# B&R Automation Studio project NAEUL004C00R13L518F00 (part 3)

### IoMap.iom - X20CP0483/IoMap.iom
```iecst
VAR_CONFIG
	::AWOpen:bModuleOK AT %IX."AutoWidth".ModuleOk;
	::AWOpen:tyParamInDriver.uiErrCode_603F AT %IW."AutoWidth".ErrorCode_603F;
	::AWOpen:tyParamOutDriver.uiCtrlword_6040 AT %QW."AutoWidth".Controlword_6040;
	::AWOpen:tyParamInDriver.uiStatword_6041 AT %IW."AutoWidth".Statusword_6041;
	::AWOpen:tyParamOutDriver.siModOfOpt_6060 AT %QB."AutoWidth".ModesOfOperation_6060;
	::AWOpen:tyParamInDriver.siModOfOptDisp_6061 AT %IB."AutoWidth".ModesOfOperationDisplay_6061;
	::AWOpen:tyParamInDriver.diActualPos_6064 AT %ID."AutoWidth".PositionActualValue_6064;
	::AWOpen:tyParamOutDriver.diTargetPos_607A AT %QD."AutoWidth".TargetPosition_607A;
	::AWOpen:tyParamOutDriver.udiMoveSpd_6081 AT %QD."AutoWidth".ProfileVelocity_6081;
	::AWOpen:tyParamOutDriver.siHmMethod_6098 AT %QB."AutoWidth".HomingMethod_6098;
	::AWOpen:tyParamInDriver.udiDigitalInputs_60FD AT %ID."AutoWidth".DigitalInputs_60FD;
	::AWOpen:tyParamOutDriver.diJogVel_60FF AT %QD."AutoWidth".TargetVelocity_60FF;
	::LifterBtm:bModuleOK AT %IX."Lifter".ModuleOk;
	::LifterBtm:tyParamInDriver.uiErrCode_603F AT %IW."Lifter".ErrorCode_603F;
	::LifterBtm:tyParamOutDriver.uiCtrlword_6040 AT %QW."Lifter".Controlword_6040;
	::LifterBtm:tyParamInDriver.uiStatword_6041 AT %IW."Lifter".Statusword_6041;
	::LifterBtm:tyParamOutDriver.siModOfOpt_6060 AT %QB."Lifter".ModesOfOperation_6060;
	::LifterBtm:tyParamInDriver.siModOfOptDisp_6061 AT %IB."Lifter".ModesOfOperationDisplay_6061;
	::LifterBtm:tyParamInDriver.diActualPos_6064 AT %ID."Lifter".PositionActualValue_6064;
	::LifterBtm:tyParamOutDriver.diTargetPos_607A AT %QD."Lifter".TargetPosition_607A;
	::LifterBtm:tyParamOutDriver.udiMoveSpd_6081 AT %QD."Lifter".ProfileVelocity_6081;
	::LifterBtm:tyParamOutDriver.siHmMethod_6098 AT %QB."Lifter".HomingMethod_6098;
	::LifterBtm:tyParamInDriver.udiDigitalInputs_60FD AT %ID."Lifter".DigitalInputs_60FD;
	::LifterBtm:tyParamOutDriver.diJogVel_60FF AT %QD."Lifter".TargetVelocity_60FF;
	::Trav:bModuleOK AT %IX."Traverser".ModuleOk;
	::Trav:tyParamInDriver.uiErrCode_603F AT %IW."Traverser".ErrorCode_603F;
	::Trav:tyParamOutDriver.uiCtrlword_6040 AT %QW."Traverser".Controlword_6040;
	::Trav:tyParamInDriver.uiStatword_6041 AT %IW."Traverser".Statusword_6041;
	::Trav:tyParamOutDriver.siModOfOpt_6060 AT %QB."Traverser".ModesOfOperation_6060;
	::Trav:tyParamInDriver.siModOfOptDisp_6061 AT %IB."Traverser".ModesOfOperationDisplay_6061;
	::Trav:tyParamInDriver.diActualPos_6064 AT %ID."Traverser".PositionActualValue_6064;
	::Trav:tyParamOutDriver.diTargetPos_607A AT %QD."Traverser".TargetPosition_607A;
	::Trav:tyParamOutDriver.udiMoveSpd_6081 AT %QD."Traverser".ProfileVelocity_6081;
	::Trav:tyParamOutDriver.siHmMethod_6098 AT %QB."Traverser".HomingMethod_6098;
	::Trav:tyParamInDriver.udiDigitalInputs_60FD AT %ID."Traverser".DigitalInputs_60FD;
	::Trav:tyParamOutDriver.diJogVel_60FF AT %QD."Traverser".TargetVelocity_60FF;
	::DInput:a_bPhysicalDI[1] AT %IX."X20DI9372".DigitalInput01;
	::DInput:a_bPhysicalDI[2] AT %IX."X20DI9372".DigitalInput02;
	::DInput:a_bPhysicalDI[3] AT %IX."X20DI9372".DigitalInput03;
	::DInput:a_bPhysicalDI[4] AT %IX."X20DI9372".DigitalInput04;
	::DInput:a_bPhysicalDI[5] AT %IX."X20DI9372".DigitalInput05;
	::DInput:a_bPhysicalDI[6] AT %IX."X20DI9372".DigitalInput06;
	::DInput:a_bPhysicalDI[7] AT %IX."X20DI9372".DigitalInput07;
	::DInput:a_bPhysicalDI[8] AT %IX."X20DI9372".DigitalInput08;
	::DInput:a_bPhysicalDI[9] AT %IX."X20DI9372".DigitalInput09;
	::DInput:a_bPhysicalDI[10] AT %IX."X20DI9372".DigitalInput10;
	::DInput:a_bPhysicalDI[11] AT %IX."X20DI9372".DigitalInput11;
	::DInput:a_bPhysicalDI[12] AT %IX."X20DI9372".DigitalInput12;
	::DInput:a_bPhysicalDI[13] AT %IX."X20DI9372a".DigitalInput01;
	::DInput:a_bPhysicalDI[14] AT %IX."X20DI9372a".DigitalInput02;
	::DInput:a_bPhysicalDI[15] AT %IX."X20DI9372a".DigitalInput03;
	::DInput:a_bPhysicalDI[16] AT %IX."X20DI9372a".DigitalInput04;
	::DInput:a_bPhysicalDI[17] AT %IX."X20DI9372a".DigitalInput05;
	::DInput:a_bPhysicalDI[18] AT %IX."X20DI9372a".DigitalInput06;
	::DInput:a_bPhysicalDI[19] AT %IX."X20DI9372a".DigitalInput07;
	::DInput:a_bPhysicalDI[20] AT %IX."X20DI9372a".DigitalInput08;
	::DInput:a_bPhysicalDI[21] AT %IX."X20DI9372a".DigitalInput09;
	::DInput:a_bPhysicalDI[22] AT %IX."X20DI9372a".DigitalInput10;
	::DInput:a_bPhysicalDI[23] AT %IX."X20DI9372a".DigitalInput11;
	::DInput:a_bPhysicalDI[24] AT %IX."X20DI9372a".DigitalInput12;
	::DInput:a_bPhysicalDI[25] AT %IX."X20DI9372b".DigitalInput01;
	::DInput:a_bPhysicalDI[26] AT %IX."X20DI9372b".DigitalInput02;
	::DInput:a_bPhysicalDI[27] AT %IX."X20DI9372b".DigitalInput03;
	::DInput:a_bPhysicalDI[28] AT %IX."X20DI9372b".DigitalInput04;
	::DInput:a_bPhysicalDI[29] AT %IX."X20DI9372b".DigitalInput05;
	::DInput:a_bPhysicalDI[30] AT %IX."X20DI9372b".DigitalInput06;
	::DInput:a_bPhysicalDI[31] AT %IX."X20DI9372b".DigitalInput07;
	::DInput:a_bPhysicalDI[32] AT %IX."X20DI9372b".DigitalInput08;
	::DInput:a_bPhysicalDI[33] AT %IX."X20DI9372b".DigitalInput09;
	::DInput:a_bPhysicalDI[34] AT %IX."X20DI9372b".DigitalInput10;
	::DInput:a_bPhysicalDI[35] AT %IX."X20DI9372b".DigitalInput11;
	::DInput:a_bPhysicalDI[36] AT %IX."X20DI9372b".DigitalInput12;
	::DInput:a_bPhysicalDI[37] AT %IX."X20DI9372c".DigitalInput01;
	::DInput:a_bPhysicalDI[38] AT %IX."X20DI9372c".DigitalInput02;
	::DInput:a_bPhysicalDI[39] AT %IX."X20DI9372c".DigitalInput03;
	::DInput:a_bPhysicalDI[40] AT %IX."X20DI9372c".DigitalInput04;
	::DInput:a_bPhysicalDI[41] AT %IX."X20DI9372c".DigitalInput05;
	::DInput:a_bPhysicalDI[42] AT %IX."X20DI9372c".DigitalInput06;
	::DInput:a_bPhysicalDI[43] AT %IX."X20DI9372c".DigitalInput07;
	::DInput:a_bPhysicalDI[44] AT %IX."X20DI9372c".DigitalInput08;
	::DInput:a_bPhysicalDI[45] AT %IX."X20DI9372c".DigitalInput09;
	::DInput:a_bPhysicalDI[46] AT %IX."X20DI9372c".DigitalInput10;
	::DInput:a_bPhysicalDI[47] AT %IX."X20DI9372c".DigitalInput11;
	::DInput:a_bPhysicalDI[48] AT %IX."X20DI9372c".DigitalInput12;
	::DOutput:a_bPhysicalDO[7] AT %QX."X20DO9321".DigitalOutput01;
	::DOutput:a_bPhysicalDO[8] AT %QX."X20DO9321".DigitalOutput02;
	::DOutput:a_bPhysicalDO[9] AT %QX."X20DO9321".DigitalOutput03;
	::DOutput:a_bPhysicalDO[10] AT %QX."X20DO9321".DigitalOutput04;
	::DOutput:a_bPhysicalDO[11] AT %QX."X20DO9321".DigitalOutput05;
	::DOutput:a_bPhysicalDO[12] AT %QX."X20DO9321".DigitalOutput06;
	::DOutput:a_bPhysicalDO[13] AT %QX."X20DO9321".DigitalOutput07;
	::DOutput:a_bPhysicalDO[14] AT %QX."X20DO9321".DigitalOutput08;
	::DOutput:a_bPhysicalDO[15] AT %QX."X20DO9321".DigitalOutput09;
	::DOutput:a_bPhysicalDO[16] AT %QX."X20DO9321".DigitalOutput10;
	::DOutput:a_bPhysicalDO[17] AT %QX."X20DO9321".DigitalOutput11;
	::DOutput:a_bPhysicalDO[18] AT %QX."X20DO9321".DigitalOutput12;
	::DOutput:a_bPhysicalDO[19] AT %QX."X20DO9321a".DigitalOutput01;
	::DOutput:a_bPhysicalDO[20] AT %QX."X20DO9321a".DigitalOutput02;
	::DOutput:a_bPhysicalDO[21] AT %QX."X20DO9321a".DigitalOutput03;
	::DOutput:a_bPhysicalDO[22] AT %QX."X20DO9321a".DigitalOutput04;
	::DOutput:a_bPhysicalDO[23] AT %QX."X20DO9321a".DigitalOutput05;
	::DOutput:a_bPhysicalDO[24] AT %QX."X20DO9321a".DigitalOutput06;
	::DOutput:a_bPhysicalDO[25] AT %QX."X20DO9321a".DigitalOutput07;
	::DOutput:a_bPhysicalDO[26] AT %QX."X20DO9321a".DigitalOutput08;
	::DOutput:a_bPhysicalDO[27] AT %QX."X20DO9321a".DigitalOutput09;
	::DOutput:a_bPhysicalDO[28] AT %QX."X20DO9321a".DigitalOutput10;
	::DOutput:a_bPhysicalDO[29] AT %QX."X20DO9321a".DigitalOutput11;
	::DOutput:a_bPhysicalDO[30] AT %QX."X20DO9321a".DigitalOutput12;
	::DOutput:a_bPhysicalDO[31] AT %QX."X20DO9321b".DigitalOutput01;
	::DOutput:a_bPhysicalDO[32] AT %QX."X20DO9321b".DigitalOutput02;
	::DOutput:a_bPhysicalDO[33] AT %QX."X20DO9321b".DigitalOutput03;
	::DOutput:a_bPhysicalDO[34] AT %QX."X20DO9321b".DigitalOutput04;
	::DOutput:a_bPhysicalDO[35] AT %QX."X20DO9321b".DigitalOutput05;
	::DOutput:a_bPhysicalDO[36] AT %QX."X20DO9321b".DigitalOutput06;
	::DOutput:a_bPhysicalDO[37] AT %QX."X20DO9321b".DigitalOutput07;
	::DOutput:a_bPhysicalDO[38] AT %QX."X20DO9321b".DigitalOutput08;
	::DOutput:a_bPhysicalDO[39] AT %QX."X20DO9321b".DigitalOutput09;
	::DOutput:a_bPhysicalDO[40] AT %QX."X20DO9321b".DigitalOutput10;
	::DOutput:a_bPhysicalDO[41] AT %QX."X20DO9321b".DigitalOutput11;
	::DOutput:a_bPhysicalDO[42] AT %QX."X20DO9321b".DigitalOutput12;
	::MagAWOpen1:bModuleOK AT %IX."Mag1_AutoWidth".ModuleOk;
	::MagAWOpen1:tyParamInDriver.uiErrCode_603F AT %IW."Mag1_AutoWidth".ErrorCode_603F;
	::MagAWOpen1:tyParamOutDriver.uiCtrlword_6040 AT %QW."Mag1_AutoWidth".Controlword_6040;
	::MagAWOpen1:tyParamInDriver.uiStatword_6041 AT %IW."Mag1_AutoWidth".Statusword_6041;
	::MagAWOpen1:tyParamOutDriver.siModOfOpt_6060 AT %QB."Mag1_AutoWidth".ModesOfOperation_6060;
	::MagAWOpen1:tyParamInDriver.siModOfOptDisp_6061 AT %IB."Mag1_AutoWidth".ModesOfOperationDisplay_6061;
	::MagAWOpen1:tyParamInDriver.diActualPos_6064 AT %ID."Mag1_AutoWidth".PositionActualValue_6064;
	::MagAWOpen1:tyParamOutDriver.diTargetPos_607A AT %QD."Mag1_AutoWidth".TargetPosition_607A;
	::MagAWOpen1:tyParamOutDriver.udiMoveSpd_6081 AT %QD."Mag1_AutoWidth".ProfileVelocity_6081;
	::MagAWOpen1:tyParamOutDriver.siHmMethod_6098 AT %QB."Mag1_AutoWidth".HomingMethod_6098;
	::MagAWOpen1:tyParamInDriver.udiDigitalInputs_60FD AT %ID."Mag1_AutoWidth".DigitalInputs_60FD;
	::MagAWOpen1:tyParamOutDriver.diJogVel_60FF AT %QD."Mag1_AutoWidth".TargetVelocity_60FF;
	::MagAWOpen2:bModuleOK AT %IX."Mag2_AutoWidth".ModuleOk;
	::MagAWOpen2:tyParamInDriver.uiErrCode_603F AT %IW."Mag2_AutoWidth".ErrorCode_603F;
	::MagAWOpen2:tyParamOutDriver.uiCtrlword_6040 AT %QW."Mag2_AutoWidth".Controlword_6040;
	::MagAWOpen2:tyParamInDriver.uiStatword_6041 AT %IW."Mag2_AutoWidth".Statusword_6041;
	::MagAWOpen2:tyParamOutDriver.siModOfOpt_6060 AT %QB."Mag2_AutoWidth".ModesOfOperation_6060;
	::MagAWOpen2:tyParamInDriver.siModOfOptDisp_6061 AT %IB."Mag2_AutoWidth".ModesOfOperationDisplay_6061;
	::MagAWOpen2:tyParamInDriver.diActualPos_6064 AT %ID."Mag2_AutoWidth".PositionActualValue_6064;
	::MagAWOpen2:tyParamOutDriver.diTargetPos_607A AT %QD."Mag2_AutoWidth".TargetPosition_607A;
	::MagAWOpen2:tyParamOutDriver.udiMoveSpd_6081 AT %QD."Mag2_AutoWidth".ProfileVelocity_6081;
	::MagAWOpen2:tyParamOutDriver.siHmMethod_6098 AT %QB."Mag2_AutoWidth".HomingMethod_6098;
	::MagAWOpen2:tyParamInDriver.udiDigitalInputs_60FD AT %ID."Mag2_AutoWidth".DigitalInputs_60FD;
	::MagAWOpen2:tyParamOutDriver.diJogVel_60FF AT %QD."Mag2_AutoWidth".TargetVelocity_60FF;
	::MagAWOpen3:bModuleOK AT %IX."Mag3_AutoWidth".ModuleOk;
	::MagAWOpen3:tyParamInDriver.uiErrCode_603F AT %IW."Mag3_AutoWidth".ErrorCode_603F;
	::MagAWOpen3:tyParamOutDriver.uiCtrlword_6040 AT %QW."Mag3_AutoWidth".Controlword_6040;
	::MagAWOpen3:tyParamInDriver.uiStatword_6041 AT %IW."Mag3_AutoWidth".Statusword_6041;
	::MagAWOpen3:tyParamOutDriver.siModOfOpt_6060 AT %QB."Mag3_AutoWidth".ModesOfOperation_6060;
	::MagAWOpen3:tyParamInDriver.siModOfOptDisp_6061 AT %IB."Mag3_AutoWidth".ModesOfOperationDisplay_6061;
	::MagAWOpen3:tyParamInDriver.diActualPos_6064 AT %ID."Mag3_AutoWidth".PositionActualValue_6064;
	::MagAWOpen3:tyParamOutDriver.diTargetPos_607A AT %QD."Mag3_AutoWidth".TargetPosition_607A;
	::MagAWOpen3:tyParamOutDriver.udiMoveSpd_6081 AT %QD."Mag3_AutoWidth".ProfileVelocity_6081;
	::MagAWOpen3:tyParamOutDriver.siHmMethod_6098 AT %QB."Mag3_AutoWidth".HomingMethod_6098;
	::MagAWOpen3:tyParamInDriver.udiDigitalInputs_60FD AT %ID."Mag3_AutoWidth".DigitalInputs_60FD;
	::MagAWOpen3:tyParamOutDriver.diJogVel_60FF AT %QD."Mag3_AutoWidth".TargetVelocity_60FF;
	::AWPushOrPu:bModuleOK AT %IX."AutoWidthPusher".ModuleOk;
	::AWPushOrPu:tyParamInDriver.uiErrCode_603F AT %IW."AutoWidthPusher".ErrorCode_603F;
	::AWPushOrPu:tyParamInDriver.uiStatword_6041 AT %IW."AutoWidthPusher".Statusword_6041;
	::AWPushOrPu:tyParamInDriver.siModOfOptDisp_6061 AT %IB."AutoWidthPusher".ModesOfOperationDisplay_6061;
	::AWPushOrPu:tyParamInDriver.diActualPos_6064 AT %ID."AutoWidthPusher".PositionActualValue_6064;
	::AWPushOrPu:tyParamInDriver.udiDigitalInputs_60FD AT %ID."AutoWidthPusher".DigitalInputs_60FD;
	::AWPushOrPu:tyParamOutDriver.uiCtrlword_6040 AT %QW."AutoWidthPusher".Controlword_6040;
	::AWPushOrPu:tyParamOutDriver.siModOfOpt_6060 AT %QB."AutoWidthPusher".ModesOfOperation_6060;
	::AWPushOrPu:tyParamOutDriver.diTargetPos_607A AT %QD."AutoWidthPusher".TargetPosition_607A;
	::AWPushOrPu:tyParamOutDriver.udiMoveSpd_6081 AT %QD."AutoWidthPusher".ProfileVelocity_6081;
	::AWPushOrPu:tyParamOutDriver.siHmMethod_6098 AT %QB."AutoWidthPusher".HomingMethod_6098;
	::AWPushOrPu:tyParamOutDriver.diJogVel_60FF AT %QD."AutoWidthPusher".TargetVelocity_60FF;
	::AWPushOrPu:tyParamOutDriver.siModOfOpt_6060 AT %QB."AutoWidthPusher".Modes_of_operation_6060;
	::AWPushOrPu:tyParamOutDriver.diTargetPos_607A AT %QD."AutoWidthPusher".Target_position_607A;
	::AWPushOrPu:tyParamOutDriver.udiMoveSpd_6081 AT %QD."AutoWidthPusher".Profile_velocity_6081;
	::AWPushOrPu:tyParamOutDriver.siHmMethod_6098 AT %QB."AutoWidthPusher".Homing_method_6098;
	::AWPushOrPu:tyParamOutDriver.diJogVel_60FF AT %QD."AutoWidthPusher".Target_velocity_60FF;
	::AWPushOrPu:tyParamInDriver.uiErrCode_603F AT %IW."AutoWidthPusher".Error_code_603F;
	::AWPushOrPu:tyParamInDriver.siModOfOptDisp_6061 AT %IB."AutoWidthPusher".Modes_of_operation_display_6061;
	::AWPushOrPu:tyParamInDriver.diActualPos_6064 AT %ID."AutoWidthPusher".Position_actual_value_6064;
	::AWPushOrPu:tyParamInDriver.udiDigitalInputs_60FD AT %ID."AutoWidthPusher".Digital_intputs_60FD;
	::PullerPush:bModuleOK AT %IX."PullerPusher".ModuleOk;
	::PullerPush:tyParamInDriver.uiErrCode_603F AT %IW."PullerPusher".ErrorCode_603F;
	::PullerPush:tyParamInDriver.uiStatword_6041 AT %IW."PullerPusher".Statusword_6041;
	::PullerPush:tyParamInDriver.siModOfOptDisp_6061 AT %IB."PullerPusher".ModesOfOperationDisplay_6061;
	::PullerPush:tyParamInDriver.udiDigitalInputs_60FD AT %ID."PullerPusher".DigitalInputs_60FD;
	::PullerPush:tyParamOutDriver.uiCtrlword_6040 AT %QW."PullerPusher".Controlword_6040;
	::PullerPush:tyParamOutDriver.siModOfOpt_6060 AT %QB."PullerPusher".ModesOfOperation_6060;
	::PullerPush:tyParamInDriver.diActualPos_6064 AT %ID."PullerPusher".PositionActualValue_6064;
	::PullerPush:tyParamOutDriver.diTargetPos_607A AT %QD."PullerPusher".TargetPosition_607A;
	::PullerPush:tyParamOutDriver.udiMoveSpd_6081 AT %QD."PullerPusher".ProfileVelocity_6081;
	::PullerPush:tyParamOutDriver.siHmMethod_6098 AT %QB."PullerPusher".HomingMethod_6098;
	::PullerPush:tyParamOutDriver.diJogVel_60FF AT %QD."PullerPusher".TargetVelocity_60FF;
	::DOutput:a_bPhysicalDO[1] AT %QX."X20DO6321".DigitalOutput01;
	::DOutput:a_bPhysicalDO[2] AT %QX."X20DO6321".DigitalOutput02;
	::DOutput:a_bPhysicalDO[3] AT %QX."X20DO6321".DigitalOutput03;
	::DOutput:a_bPhysicalDO[4] AT %QX."X20DO6321".DigitalOutput04;
	::DOutput:a_bPhysicalDO[5] AT %QX."X20DO6321".DigitalOutput05;
	::DOutput:a_bPhysicalDO[6] AT %QX."X20DO6321".DigitalOutput06;
END_VAR
```

## Configuration 3Mag_UL_MagAW_SOT

CPU X20CP0483, AutomationRuntime B4.82, Build 4.1.2, Safety 0.0, Vc V4.72.1

### Task classes (Cpu.sw)
```
Cyclic#1 (cycle 10000 us, tolerance 10000 us):
  DInput <- DInput.DInput.prg
  DOutput <- DOutput.DOutput.prg
Cyclic#2 (cycle 20000 us, tolerance 20000 us):
  PshrConv <- Conv.PshrConv.prg
  MagConv2Cl <- MagConv_LiftnTrav.MagConv2Clp1.prg
  MagConv2C1 <- MagConv_LiftnTrav.MagConv2Clp2.prg
  MagConv2C2 <- MagConv_LiftnTrav.MagConv2Clp3.prg
  MtrPshr <- MtrPshr.MtrPshr.prg
  PullerPush <- CANOpenServo.PullerPusher.PullerPusher.prg
Cyclic#3 (cycle 50000 us, tolerance 50000 us):
  UI <- UI.UI.prg
  Startup <- Startup.Startup.prg
  General <- General.General.prg
  UsrFolder <- UsrFolder.UsrFolder.prg
  LibVer <- LibVer.LibVer.prg
  Time <- Time.Time.prg
  HWInfo <- HWInfo.HWInfo.prg
  TLBuz <- TLBuz.TLBuz.prg
  Alarm <- Alarm.Alarm.prg
  RstErr <- RstErr.RstErr.prg
  ProdRcp <- ProdRcp.ProdRcp.prg
  MpProdRcp <- MpProdRcp.MpProdRcp.prg
  MagRcp <- MagRcp.MagRcp.prg
  McParam <- McParam.McParam.prg
  NtParam <- NtParam.NtParam.prg
  UsrMgmt <- UsrMgmt.UsrMgmt.prg
  OvenInfoA <- OvenInfo.OvenInfoA.prg
  OvenInfoB <- OvenInfo.OvenInfoB.prg
  Buffer1 <- Buffer.Buffer1.prg
  Buffer2 <- Buffer.Buffer2.prg
  Buffer3 <- Buffer.Buffer3.prg
  BufferMagA <- Buffer.BufferMagA.prg
  BufferMagB <- Buffer.BufferMagB.prg
  USSMEMAA <- SMEMA.USSMEMAA.prg
  USSMEMAB <- SMEMA.USSMEMAB.prg
  USSMEMA1 <- SMEMA.USSMEMA1.prg
  USSMEMA2 <- SMEMA.USSMEMA2.prg
  USSMEMA3 <- SMEMA.USSMEMA3.prg
  DSSMEMA1 <- SMEMA.DSSMEMA1.prg
  DSSMEMA2 <- SMEMA.DSSMEMA2.prg
  DSSMEMA3 <- SMEMA.DSSMEMA3.prg
  Pneu2SenIn <- Pneu.Pneu2SenInShutter.prg
  Pneu2SenOu <- Pneu.Pneu2SenOutShutter.prg
  PneuNoSenS <- Pneu.PneuNoSenStopperA.prg
  PneuNoSen1 <- Pneu.PneuNoSenStopperB.prg
  PneuNoSen2 <- Pneu.PneuNoSenStopperC.prg
  Pneu2SenSe <- Pneu.Pneu2SenSelClamp1.prg
  Pneu2SenS1 <- Pneu.Pneu2SenSelClamp2.prg
  Pneu2SenS2 <- Pneu.Pneu2SenSelClamp3.prg
  Pneu2SenMa <- Pneu.Pneu2SenMag1SafetyBar.prg
  Pneu2SenM1 <- Pneu.Pneu2SenMag2SafetyBar.prg
  Pneu2SenM2 <- Pneu.Pneu2SenMag3SafetyBar.prg
  Pneu2SenM3 <- Pneu.Pneu2SenMag1AWEngage.prg
  Pneu2SenM4 <- Pneu.Pneu2SenMag2AWEngage.prg
  Pneu2SenM5 <- Pneu.Pneu2SenMag3AWEngage.prg
  PneuNoSenT <- Pneu.MagConv_Stopper.PneuNoSenTopEntStpr.prg
  PneuNoSen3 <- Pneu.MagConv_Stopper.PneuNoSenTopMidStpr.prg
  PneuNoSen4 <- Pneu.MagConv_Stopper.PneuNoSenTopExtStpr.prg
  PneuNoSenB <- Pneu.MagConv_Stopper.PneuNoSenBtmMidStpr.prg
  PneuNoSen5 <- Pneu.MagConv_Stopper.PneuNoSenBtmExtStpr.prg
  PneuNoSen6 <- Pneu.MagConv_Stopper.PneuNoSenTopEntStpr2.prg
  PneuNoSen7 <- Pneu.MagConv_Stopper.PneuNoSenTopMidStpr2.prg
  PneuNoSen8 <- Pneu.MagConv_Stopper.PneuNoSenTopExtStpr2.prg
  PneuNoSen9 <- Pneu.MagConv_Stopper.PneuNoSenBtmMidStpr2.prg
  PneuNoSe10 <- Pneu.MagConv_Stopper.PneuNoSenBtmExtStpr2.prg
  Pneu2SenO1 <- Pneu.Pneu2SenOutShutter2.prg
  Pneu2SenO2 <- Pneu.Pneu2SenOutShutter3.prg
  InMagConv <- MagConv_TopBtm.InMagConv.prg
  OutMagConv <- MagConv_TopBtm.OutMagConv.prg
  LifterMagC <- MagConv_TopBtm.LifterMagConv.prg
  InMagConv2 <- MagConv_TopBtm.InMagConv2.prg
  OutMagCon1 <- MagConv_TopBtm.OutMagConv2.prg
  LifterMag1 <- MagConv_TopBtm.LifterMagConv2.prg
  AWOpen <- CANOpenServo.AW.AWOpen.prg
  AWPushOrPu <- CANOpenServo.AW.AWPushOrPuller.prg
  Trav <- CANOpenServo.Trav.Trav.prg
  LifterBtm <- CANOpenServo.Lifter.LifterBtm.prg
  Lifter2 <- CANOpenServo.Lifter.Lifter2.prg
  MagAWOpen1 <- CANOpenServo.MagAW.MagAWOpen1.prg
  MagAWOpen2 <- CANOpenServo.MagAW.MagAWOpen2.prg
  MagAWOpen3 <- CANOpenServo.MagAW.MagAWOpen3.prg
  Hermes <- Hermes.Hermes.prg
  USHermesA <- Hermes.USHermesA.prg
  USHermesB <- Hermes.USHermesB.prg
  RmtHermes <- Hermes.RmtHermes.prg
  SvyHermes <- Hermes.SvyHermes.prg
  LFLeader <- LF.LFLeader.prg
  LFFollower <- LF.LFFollower.prg
  Follower1 <- LF.Follower1.prg
  Follower2 <- LF.Follower2.prg
  LCS <- LCS.LCS.prg
  LCSMngRcp <- LCS.LCSMngRcp.prg
  LCSLF <- LCS.LCSLF.prg
  Ops <- Operations.Ops.prg
  OpsTravLif <- Operations.OpsTravLifUL.prg
  OpsMagConv <- Operations.MagConv_StationaryPlat.OpsMagConvUL1.prg
  OpsMagCon1 <- Operations.MagConv_StationaryPlat.OpsMagConvUL2.prg
  OpsMagCon2 <- Operations.MagConv_StationaryPlat.OpsMagConvUL3.prg
  OpsLifMagU <- Operations.OpsLifMagUL.prg
  OpsInMagCo <- Operations.MultiMag_InOutMagazineConv.OpsInMagConv.prg
  OpsOutMagC <- Operations.MultiMag_InOutMagazineConv.OpsOutMagConv.prg
  OpsMagCon3 <- Operations.MultiMag_InOutMagazineConv.OpsMagConvStpr.prg
  OpsMagCon4 <- Operations.MultiMag_InOutMagazineConv.OpsMagConvStpr2.prg
  AGV <- AGVCom.AGV.prg
  AGV1 <- AGVCom.AGV1.prg
  AGV2 <- AGVCom.AGV2.prg
  AGV3 <- AGVCom.AGV3.prg
  Simu <- Simulation.Simu.prg
  Simu1 <- Simulation.Simu1.prg
  Machine <- Machine.Machine.prg
  USSOT1 <- SOT.USSOT1.prg
  DSSOT1 <- SOT.DSSOT1.prg
  USSOT2 <- SOT.USSOT2.prg
  DSSOT2 <- SOT.DSSOT2.prg
  USSOT3 <- SOT.USSOT3.prg
  DSSOT3 <- SOT.DSSOT3.prg
  TCP <- TCP.TCP.prg
  TCPTop <- TCP.TCPTop.prg
  TCPBtm <- TCP.TCPBtm.prg
  OpCon <- OpCon.OpCon.prg
DataObjects: Acp10sys
VcDataObjects: Visu <- UI.Visu.dob
Binaries: vcfntttf, arialbi, vccbmp, vcshared, vcpdvnc, vccshape, vcfile, vcgclass, arial, vcchspot, vcmgr, arialxsr, vccslider, vcdsint, vccbtn, vcdsloc, vccovl, vccpopup, vccline, vcctext, vcalarm, vcbclass, vccbar, visvc, udbdef, vcrt, vccnum, vccstr, Visu03, vccddbox, arialbd, vcpdsw, vcnet, TCData, Visu02, Visu01, vctcal, vccdt, vcpfgen, vccalarm, arsvcreg, acp10cfg, Acp10map, arconfig, asfw, iomap, Role, ashwd, ashwac, sysconf, User, Config, vcpfar00, OpcUaMap
Libraries: standard, runtime, astime, asstring, operator, AsIecCon, AsCANopen, visapi, FileIO, AsIODiag, AsMem, dvframe, AsOpcUac, AsARCfg, sys_lib, AsTCP, AsFltGen, brsystem, MpRecipe, MpBase, MpCom, NtBuffer, NtConv, NtFileIO, NtLogFile, NtMem, NtMessage, NtOvenInfo, NtPneu, NtRS232, NtSMEMA, NtTCP, NtTLBuz, NtVersion, NtSOT, NtLF, NtMotion, NtRecipe, NtGeneral, NtUI, Acp10man, Acp10par, NcGlobal, NtHermes, dataobj, vcresman, powerlnk, NtOpConXML
```

### Hardware
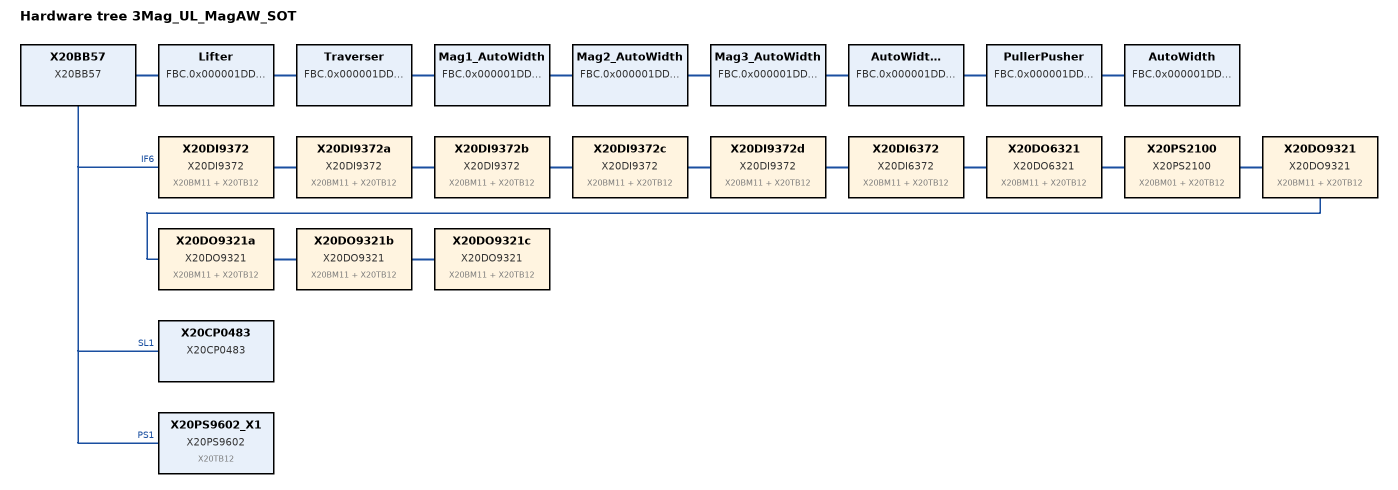
```
AutoWidth : FBC.0x000001DD.0x00000001.NUTEK_DELTA_EDS_V101 v1.0 (OrderNumber=NUTEK_DELTA_V101)  [CAN1 -> PullerPusher.CAN2 (NodeNumber=16)]
AutoWidthPusher : FBC.0x000001DD.0x00000001.NUTEK_DELTA_EDS_V101 v1.0 (OrderNumber=NUTEK_DELTA_V101)  [CAN1 -> Mag3_AutoWidth.CAN2]
Lifter : FBC.0x000001DD.0x00000001.NUTEK_DELTA_EDS_V101 v1.0 (OrderNumber=NUTEK_DELTA_V101)  [CAN1 -> X20BB57.IF7 (NodeNumber=17)]
  p210c_parametervalue = 300
Mag1_AutoWidth : FBC.0x000001DD.0x00000001.NUTEK_DELTA_EDS_V101 v1.0 (OrderNumber=NUTEK_DELTA_V101)  [CAN1 -> Traverser.CAN2 (NodeNumber=19)]
  p210c_parametervalue = 60
  p210d_parametervalue = 60
  p210e_parametervalue = 60
  p220a_parametervalue = 0x0001
  p220c_parametervalue = 0x0016
  p220d_parametervalue = 0x0017
Mag2_AutoWidth : FBC.0x000001DD.0x00000001.NUTEK_DELTA_EDS_V101 v1.0 (OrderNumber=NUTEK_DELTA_V101)  [CAN1 -> Mag1_AutoWidth.CAN2]
  p210c_parametervalue = 60
  p210d_parametervalue = 60
  p210e_parametervalue = 60
  p220a_parametervalue = 0x0001
  p220c_parametervalue = 0x0016
  p220d_parametervalue = 0x0017
Mag3_AutoWidth : FBC.0x000001DD.0x00000001.NUTEK_DELTA_EDS_V101 v1.0 (OrderNumber=NUTEK_DELTA_V101)  [CAN1 -> Mag2_AutoWidth.CAN2]
  p210c_parametervalue = 60
  p210d_parametervalue = 60
  p210e_parametervalue = 60
  p220a_parametervalue = 0x0001
  p220c_parametervalue = 0x0016
  p220d_parametervalue = 0x0017
PullerPusher : FBC.0x000001DD.0x00000001.NUTEK_DELTA_EDS_V101 v1.0 (OrderNumber=NUTEK_DELTA_V101)  [CAN1 -> AutoWidthPusher.CAN2]
Traverser : FBC.0x000001DD.0x00000001.NUTEK_DELTA_EDS_V101 v1.0 (OrderNumber=NUTEK_DELTA_V101)  [CAN1 -> Lifter.CAN2]
X20BB57 : X20BB57 v1.1.1.0
  Connector IF1:
    Baudrate = 9600
    Parity = N
  Connector IF7:
    Baudrate = 1000000
    ActivateCanOpen = 1
    p100c_parametervalue = 1000
    p100d_parametervalue = 3
X20BM01 : X20BM01 v2.1.0.0  [X2X1 -> X20BM11e.X2X2]
X20BM11 : X20BM11 v1.0.0.1  [X2X1 -> X20BB57.IF6]
X20BM11a : X20BM11 v1.0.0.1  [X2X1 -> X20BM11.X2X2]
X20BM11b : X20BM11 v1.0.0.1  [X2X1 -> X20BM11a.X2X2]
X20BM11c : X20BM11 v1.0.0.1  [X2X1 -> X20BM11b.X2X2]
X20BM11d : X20BM11 v1.0.0.1  [X2X1 -> X20BM11c.X2X2]
X20BM11e : X20BM11 v1.0.0.1  [X2X1 -> X20BM11i.X2X2]
X20BM11f : X20BM11 v1.0.0.1  [X2X1 -> X20BM01.X2X2]
X20BM11g : X20BM11 v1.0.0.1  [X2X1 -> X20BM11f.X2X2]
X20BM11h : X20BM11 v1.0.0.1  [X2X1 -> X20BM11g.X2X2]
X20BM11i : X20BM11 v1.0.0.1  [X2X1 -> X20BM11d.X2X2]
X20BM11j : X20BM11 v1.0.0.1  [X2X1 -> X20BM11h.X2X2]
X20CP0483 : X20CP0483 v1.2.1.0  [SL -> X20BB57.SL1]
  Connector IF2:
    ActivateDevice = 1
    Mode = Manual
    InternetAddress = 192.168.0.6
    SubnetMask = 255.255.255.0
    InaNodeNumber = 6
    Vnc1
    VncVcObjectName1 = Visu
    VncKeyMappingFile1 = 
    VncMaxConnections1 = 3
    VncRefreshRate1 = 100
    ActivateSnmp = 2
  ConfigurationID = NAEUL004
  UserPartitionSize = 150
  VolatileGlobalPvSize = 80000
  EnableUsbRemoteInstall = 1
  TimerDeviceType = SWIOTIMER
  Cyclic1Duration = 10000
  Cyclic1Tolerance = 10000
  Cyclic2Duration = 20000
  Cyclic2Tolerance = 20000
  Cyclic3Duration = 50000
  Cyclic3Tolerance = 50000
  Cyclic4Duration = 10000
  Cyclic4Tolerance = 10000
  Cyclic5Duration = 200000
  Cyclic5Tolerance = 200000
  Cyclic6Duration = 500000
  Cyclic6Tolerance = 500000
  Cyclic7Duration = 1000000
  Cyclic7Tolerance = 1000000
  Cyclic8Duration = 10000
  Cyclic8Tolerance = 10000
  FileDevice1
  FileDeviceName1 = F
  FileDevicePath1 = F:
  FileDevice2
  FileDeviceName2 = User
  FileDevicePath2 = F:\User
  FileDevice3
  FileDeviceName3 = Private
  FileDevicePath3 = F:\Private
  FileDevice4
  FileDeviceName4 = CustomerUser
  FileDevicePath4 = F:\User\UserMgmt
  FileDevice5
  FileDeviceName5 = ProdRcp
  FileDevicePath5 = F:\User\ProductRecipe
  FileDevice6
  FileDeviceName6 = MagRcp
  FileDevicePath6 = F:\User\MagazineRecipe
  FileDevice7
  FileDeviceName7 = Alarm
  FileDevicePath7 = F:\User\Alarm
  FileDevice8
  FileDeviceName8 = McParam
  FileDevicePath8 = F:\User\MachineParameter
  FileDevice9
  FileDeviceName9 = NtParam
  FileDevicePath9 = F:\Private\NutekParameter
  FileDevice10
  FileDeviceName10 = LibVer
  FileDevicePath10 = F:\User\LibrariesVersion
  FileDevice11
  FileDeviceName11 = Retain
  FileDevicePath11 = F:\User\Retain
  FileDevice12
  FileDeviceName12 = Log
  FileDevicePath12 = F:\User\Log
  FileDevice13
  FileDeviceName13 = LCS
  FileDevicePath13 = F:\User\LCS
  FileDevice14
  FileDeviceName14 = MpProdRcp
  FileDevicePath14 = F:\User\ProductRecipeXml
  FileDevice15
  FileDeviceName15 = MpNtParam
  FileDevicePath15 = F:\Private\NutekParameterXml
  FtpUser1
  FtpUsername1 = NTAFTP
  FtpUserPassword1 = +UZ5u8Axw7KkkY4oM/r7wOOfB5oWHxpSY6r3j++jJso=  // NTA4BH
  FtpUserSalt1 = c0Alfi1W
  FTPAccessRight1 = 0
  FTPdevice1 = ALL
  FtpUser2
  FtpUsername2 = admin
  FtpUserPassword2 = mW+qRsE1LOSFDAB60rBJwb9dZ7uQUIuoHZp04C+x5XU=  // admin
  FtpUserSalt2 = Nr9+IHjr
  FTPAccessRight2 = 0
  FTPMSPartition2 = SYSTEM
  FTPMSpath2 = User
  FtpUser3
  FtpUsername3 = LCS
  FtpUserPassword3 = W4lkF6NjcyaB1sRdLwIoSAlqHoAE4GimWQdq7pKTzbA=  // LCS
  FtpUserSalt3 = f3H7b7h0
  FTPMSPartition3 = SYSTEM
  FTPMSpath3 = User\LCS
  ActivateOpcUa = 1
  OpcUaInformationModels_PV_Version = 1
X20DI6372 : X20DI6372 v1.1.0.0  [SS1 -> X20TB12k.SS; SL -> X20BM11i.SL1]
X20DI9372 : X20DI9372 v1.1.0.0  [SS1 -> X20TB12a.SS; SL -> X20BM11.SL1]
X20DI9372a : X20DI9372 v1.1.0.0  [SS1 -> X20TB12b.SS; SL -> X20BM11a.SL1]
X20DI9372b : X20DI9372 v1.1.0.0  [SS1 -> X20TB12c.SS; SL -> X20BM11b.SL1]
X20DI9372c : X20DI9372 v1.1.0.0  [SS1 -> X20TB12d.SS; SL -> X20BM11c.SL1]
X20DI9372d : X20DI9372 v1.1.0.0  [SS1 -> X20TB12e.SS; SL -> X20BM11d.SL1]
X20DO6321 : X20DO6321 v1.1.0.0  [SS1 -> X20TB12f.SS; SL -> X20BM11e.SL1]
X20DO9321 : X20DO9321 v1.1.0.0  [SS1 -> X20TB12h.SS; SL -> X20BM11f.SL1]
X20DO9321a : X20DO9321 v1.1.0.0  [SS1 -> X20TB12i.SS; SL -> X20BM11g.SL1]
X20DO9321b : X20DO9321 v1.1.0.0  [SS1 -> X20TB12j.SS; SL -> X20BM11h.SL1]
X20DO9321c : X20DO9321 v1.1.0.0  [SS1 -> X20TB12l.SS; SL -> X20BM11j.SL1]
X20PS2100 : X20PS2100 v1.2.0.0  [SS1 -> X20TB12g.SS; SL -> X20BM01.SL1]
X20PS9602_X1 : X20PS9602 v1.0.2.0  [PS -> X20BB57.PS1; SS1 -> X20TB12.SS]
X20TB12 : X20TB12 v1.0.0.0
X20TB12a : X20TB12 v1.0.0.0
X20TB12b : X20TB12 v1.0.0.0
X20TB12c : X20TB12 v1.0.0.0
X20TB12d : X20TB12 v1.0.0.0
X20TB12e : X20TB12 v1.0.0.0
X20TB12f : X20TB12 v1.0.0.0
X20TB12g : X20TB12 v1.0.0.0
X20TB12h : X20TB12 v1.0.0.0
X20TB12i : X20TB12 v1.0.0.0
X20TB12j : X20TB12 v1.0.0.0
X20TB12k : X20TB12 v1.0.0.0
X20TB12l : X20TB12 v1.0.0.0
```

### IoMap.iom - X20CP0483/IoMap.iom
```iecst
VAR_CONFIG
	::AWOpen:bModuleOK AT %IX."AutoWidth".ModuleOk;
	::AWOpen:tyParamInDriver.uiErrCode_603F AT %IW."AutoWidth".ErrorCode_603F;
	::AWOpen:tyParamOutDriver.uiCtrlword_6040 AT %QW."AutoWidth".Controlword_6040;
	::AWOpen:tyParamInDriver.uiStatword_6041 AT %IW."AutoWidth".Statusword_6041;
	::AWOpen:tyParamOutDriver.siModOfOpt_6060 AT %QB."AutoWidth".ModesOfOperation_6060;
	::AWOpen:tyParamInDriver.siModOfOptDisp_6061 AT %IB."AutoWidth".ModesOfOperationDisplay_6061;
	::AWOpen:tyParamInDriver.diActualPos_6064 AT %ID."AutoWidth".PositionActualValue_6064;
	::AWOpen:tyParamOutDriver.diTargetPos_607A AT %QD."AutoWidth".TargetPosition_607A;
	::AWOpen:tyParamOutDriver.udiMoveSpd_6081 AT %QD."AutoWidth".ProfileVelocity_6081;
	::AWOpen:tyParamOutDriver.siHmMethod_6098 AT %QB."AutoWidth".HomingMethod_6098;
	::AWOpen:tyParamInDriver.udiDigitalInputs_60FD AT %ID."AutoWidth".DigitalInputs_60FD;
	::AWOpen:tyParamOutDriver.diJogVel_60FF AT %QD."AutoWidth".TargetVelocity_60FF;
	::LifterBtm:bModuleOK AT %IX."Lifter".ModuleOk;
	::LifterBtm:tyParamInDriver.uiErrCode_603F AT %IW."Lifter".ErrorCode_603F;
	::LifterBtm:tyParamOutDriver.uiCtrlword_6040 AT %QW."Lifter".Controlword_6040;
	::LifterBtm:tyParamInDriver.uiStatword_6041 AT %IW."Lifter".Statusword_6041;
	::LifterBtm:tyParamOutDriver.siModOfOpt_6060 AT %QB."Lifter".ModesOfOperation_6060;
	::LifterBtm:tyParamInDriver.siModOfOptDisp_6061 AT %IB."Lifter".ModesOfOperationDisplay_6061;
	::LifterBtm:tyParamInDriver.diActualPos_6064 AT %ID."Lifter".PositionActualValue_6064;
	::LifterBtm:tyParamOutDriver.diTargetPos_607A AT %QD."Lifter".TargetPosition_607A;
	::LifterBtm:tyParamOutDriver.udiMoveSpd_6081 AT %QD."Lifter".ProfileVelocity_6081;
	::LifterBtm:tyParamOutDriver.siHmMethod_6098 AT %QB."Lifter".HomingMethod_6098;
	::LifterBtm:tyParamInDriver.udiDigitalInputs_60FD AT %ID."Lifter".DigitalInputs_60FD;
	::LifterBtm:tyParamOutDriver.diJogVel_60FF AT %QD."Lifter".TargetVelocity_60FF;
	::Trav:bModuleOK AT %IX."Traverser".ModuleOk;
	::Trav:tyParamInDriver.uiErrCode_603F AT %IW."Traverser".ErrorCode_603F;
	::Trav:tyParamOutDriver.uiCtrlword_6040 AT %QW."Traverser".Controlword_6040;
	::Trav:tyParamInDriver.uiStatword_6041 AT %IW."Traverser".Statusword_6041;
	::Trav:tyParamOutDriver.siModOfOpt_6060 AT %QB."Traverser".ModesOfOperation_6060;
	::Trav:tyParamInDriver.siModOfOptDisp_6061 AT %IB."Traverser".ModesOfOperationDisplay_6061;
	::Trav:tyParamInDriver.diActualPos_6064 AT %ID."Traverser".PositionActualValue_6064;
	::Trav:tyParamOutDriver.diTargetPos_607A AT %QD."Traverser".TargetPosition_607A;
	::Trav:tyParamOutDriver.udiMoveSpd_6081 AT %QD."Traverser".ProfileVelocity_6081;
	::Trav:tyParamOutDriver.siHmMethod_6098 AT %QB."Traverser".HomingMethod_6098;
	::Trav:tyParamInDriver.udiDigitalInputs_60FD AT %ID."Traverser".DigitalInputs_60FD;
	::Trav:tyParamOutDriver.diJogVel_60FF AT %QD."Traverser".TargetVelocity_60FF;
	::DInput:a_bPhysicalDI[1] AT %IX."X20DI9372".DigitalInput01;
	::DInput:a_bPhysicalDI[2] AT %IX."X20DI9372".DigitalInput02;
	::DInput:a_bPhysicalDI[3] AT %IX."X20DI9372".DigitalInput03;
	::DInput:a_bPhysicalDI[4] AT %IX."X20DI9372".DigitalInput04;
	::DInput:a_bPhysicalDI[5] AT %IX."X20DI9372".DigitalInput05;
	::DInput:a_bPhysicalDI[6] AT %IX."X20DI9372".DigitalInput06;
	::DInput:a_bPhysicalDI[7] AT %IX."X20DI9372".DigitalInput07;
	::DInput:a_bPhysicalDI[8] AT %IX."X20DI9372".DigitalInput08;
	::DInput:a_bPhysicalDI[9] AT %IX."X20DI9372".DigitalInput09;
	::DInput:a_bPhysicalDI[10] AT %IX."X20DI9372".DigitalInput10;
	::DInput:a_bPhysicalDI[11] AT %IX."X20DI9372".DigitalInput11;
	::DInput:a_bPhysicalDI[12] AT %IX."X20DI9372".DigitalInput12;
	::DInput:a_bPhysicalDI[13] AT %IX."X20DI9372a".DigitalInput01;
	::DInput:a_bPhysicalDI[14] AT %IX."X20DI9372a".DigitalInput02;
	::DInput:a_bPhysicalDI[15] AT %IX."X20DI9372a".DigitalInput03;
	::DInput:a_bPhysicalDI[16] AT %IX."X20DI9372a".DigitalInput04;
	::DInput:a_bPhysicalDI[17] AT %IX."X20DI9372a".DigitalInput05;
	::DInput:a_bPhysicalDI[18] AT %IX."X20DI9372a".DigitalInput06;
	::DInput:a_bPhysicalDI[19] AT %IX."X20DI9372a".DigitalInput07;
	::DInput:a_bPhysicalDI[20] AT %IX."X20DI9372a".DigitalInput08;
	::DInput:a_bPhysicalDI[21] AT %IX."X20DI9372a".DigitalInput09;
	::DInput:a_bPhysicalDI[22] AT %IX."X20DI9372a".DigitalInput10;
	::DInput:a_bPhysicalDI[23] AT %IX."X20DI9372a".DigitalInput11;
	::DInput:a_bPhysicalDI[24] AT %IX."X20DI9372a".DigitalInput12;
	::DInput:a_bPhysicalDI[25] AT %IX."X20DI9372b".DigitalInput01;
	::DInput:a_bPhysicalDI[26] AT %IX."X20DI9372b".DigitalInput02;
	::DInput:a_bPhysicalDI[27] AT %IX."X20DI9372b".DigitalInput03;
	::DInput:a_bPhysicalDI[28] AT %IX."X20DI9372b".DigitalInput04;
	::DInput:a_bPhysicalDI[29] AT %IX."X20DI9372b".DigitalInput05;
	::DInput:a_bPhysicalDI[30] AT %IX."X20DI9372b".DigitalInput06;
	::DInput:a_bPhysicalDI[31] AT %IX."X20DI9372b".DigitalInput07;
	::DInput:a_bPhysicalDI[32] AT %IX."X20DI9372b".DigitalInput08;
	::DInput:a_bPhysicalDI[33] AT %IX."X20DI9372b".DigitalInput09;
	::DInput:a_bPhysicalDI[34] AT %IX."X20DI9372b".DigitalInput10;
	::DInput:a_bPhysicalDI[35] AT %IX."X20DI9372b".DigitalInput11;
	::DInput:a_bPhysicalDI[36] AT %IX."X20DI9372b".DigitalInput12;
	::DInput:a_bPhysicalDI[37] AT %IX."X20DI9372c".DigitalInput01;
	::DInput:a_bPhysicalDI[38] AT %IX."X20DI9372c".DigitalInput02;
	::DInput:a_bPhysicalDI[39] AT %IX."X20DI9372c".DigitalInput03;
	::DInput:a_bPhysicalDI[40] AT %IX."X20DI9372c".DigitalInput04;
	::DInput:a_bPhysicalDI[41] AT %IX."X20DI9372c".DigitalInput05;
	::DInput:a_bPhysicalDI[42] AT %IX."X20DI9372c".DigitalInput06;
	::DInput:a_bPhysicalDI[43] AT %IX."X20DI9372c".DigitalInput07;
	::DInput:a_bPhysicalDI[44] AT %IX."X20DI9372c".DigitalInput08;
	::DInput:a_bPhysicalDI[45] AT %IX."X20DI9372c".DigitalInput09;
	::DInput:a_bPhysicalDI[46] AT %IX."X20DI9372c".DigitalInput10;
	::DInput:a_bPhysicalDI[47] AT %IX."X20DI9372c".DigitalInput11;
	::DInput:a_bPhysicalDI[48] AT %IX."X20DI9372c".DigitalInput12;
	::DInput:a_bPhysicalDI[49] AT %IX."X20DI9372d".DigitalInput01;
	::DInput:a_bPhysicalDI[50] AT %IX."X20DI9372d".DigitalInput02;
	::DInput:a_bPhysicalDI[51] AT %IX."X20DI9372d".DigitalInput03;
	::DInput:a_bPhysicalDI[52] AT %IX."X20DI9372d".DigitalInput04;
	::DInput:a_bPhysicalDI[53] AT %IX."X20DI9372d".DigitalInput05;
	::DInput:a_bPhysicalDI[54] AT %IX."X20DI9372d".DigitalInput06;
	::DInput:a_bPhysicalDI[55] AT %IX."X20DI9372d".DigitalInput07;
	::DInput:a_bPhysicalDI[56] AT %IX."X20DI9372d".DigitalInput08;
	::DInput:a_bPhysicalDI[57] AT %IX."X20DI9372d".DigitalInput09;
	::DInput:a_bPhysicalDI[58] AT %IX."X20DI9372d".DigitalInput10;
	::DInput:a_bPhysicalDI[59] AT %IX."X20DI9372d".DigitalInput11;
	::DInput:a_bPhysicalDI[60] AT %IX."X20DI9372d".DigitalInput12;
	::DOutput:a_bPhysicalDO[1] AT %QX."X20DO6321".DigitalOutput01;
	::DOutput:a_bPhysicalDO[2] AT %QX."X20DO6321".DigitalOutput02;
	::DOutput:a_bPhysicalDO[3] AT %QX."X20DO6321".DigitalOutput03;
	::DOutput:a_bPhysicalDO[4] AT %QX."X20DO6321".DigitalOutput04;
	::DOutput:a_bPhysicalDO[5] AT %QX."X20DO6321".DigitalOutput05;
	::DOutput:a_bPhysicalDO[6] AT %QX."X20DO6321".DigitalOutput06;
	::DOutput:a_bPhysicalDO[7] AT %QX."X20DO9321".DigitalOutput01;
	::DOutput:a_bPhysicalDO[8] AT %QX."X20DO9321".DigitalOutput02;
	::DOutput:a_bPhysicalDO[9] AT %QX."X20DO9321".DigitalOutput03;
	::DOutput:a_bPhysicalDO[10] AT %QX."X20DO9321".DigitalOutput04;
	::DOutput:a_bPhysicalDO[11] AT %QX."X20DO9321".DigitalOutput05;
	::DOutput:a_bPhysicalDO[12] AT %QX."X20DO9321".DigitalOutput06;
	::DOutput:a_bPhysicalDO[13] AT %QX."X20DO9321".DigitalOutput07;
	::DOutput:a_bPhysicalDO[14] AT %QX."X20DO9321".DigitalOutput08;
	::DOutput:a_bPhysicalDO[15] AT %QX."X20DO9321".DigitalOutput09;
	::DOutput:a_bPhysicalDO[16] AT %QX."X20DO9321".DigitalOutput10;
	::DOutput:a_bPhysicalDO[17] AT %QX."X20DO9321".DigitalOutput11;
	::DOutput:a_bPhysicalDO[18] AT %QX."X20DO9321".DigitalOutput12;
	::DOutput:a_bPhysicalDO[19] AT %QX."X20DO9321a".DigitalOutput01;
	::DOutput:a_bPhysicalDO[20] AT %QX."X20DO9321a".DigitalOutput02;
	::DOutput:a_bPhysicalDO[21] AT %QX."X20DO9321a".DigitalOutput03;
	::DOutput:a_bPhysicalDO[22] AT %QX."X20DO9321a".DigitalOutput04;
	::DOutput:a_bPhysicalDO[23] AT %QX."X20DO9321a".DigitalOutput05;
	::DOutput:a_bPhysicalDO[24] AT %QX."X20DO9321a".DigitalOutput06;
	::DOutput:a_bPhysicalDO[25] AT %QX."X20DO9321a".DigitalOutput07;
	::DOutput:a_bPhysicalDO[26] AT %QX."X20DO9321a".DigitalOutput08;
	::DOutput:a_bPhysicalDO[27] AT %QX."X20DO9321a".DigitalOutput09;
	::DOutput:a_bPhysicalDO[28] AT %QX."X20DO9321a".DigitalOutput10;
	::DOutput:a_bPhysicalDO[29] AT %QX."X20DO9321a".DigitalOutput11;
	::DOutput:a_bPhysicalDO[30] AT %QX."X20DO9321a".DigitalOutput12;
	::DOutput:a_bPhysicalDO[31] AT %QX."X20DO9321b".DigitalOutput01;
	::DOutput:a_bPhysicalDO[32] AT %QX."X20DO9321b".DigitalOutput02;
	::DOutput:a_bPhysicalDO[33] AT %QX."X20DO9321b".DigitalOutput03;
	::DOutput:a_bPhysicalDO[34] AT %QX."X20DO9321b".DigitalOutput04;
	::DOutput:a_bPhysicalDO[35] AT %QX."X20DO9321b".DigitalOutput05;
	::DOutput:a_bPhysicalDO[36] AT %QX."X20DO9321b".DigitalOutput06;
	::DOutput:a_bPhysicalDO[37] AT %QX."X20DO9321b".DigitalOutput07;
	::DOutput:a_bPhysicalDO[38] AT %QX."X20DO9321b".DigitalOutput08;
	::DOutput:a_bPhysicalDO[39] AT %QX."X20DO9321b".DigitalOutput09;
	::DOutput:a_bPhysicalDO[40] AT %QX."X20DO9321b".DigitalOutput10;
	::DOutput:a_bPhysicalDO[41] AT %QX."X20DO9321b".DigitalOutput11;
	::DOutput:a_bPhysicalDO[42] AT %QX."X20DO9321b".DigitalOutput12;
	::MagAWOpen1:bModuleOK AT %IX."Mag1_AutoWidth".ModuleOk;
	::MagAWOpen1:tyParamInDriver.uiErrCode_603F AT %IW."Mag1_AutoWidth".ErrorCode_603F;
	::MagAWOpen1:tyParamOutDriver.uiCtrlword_6040 AT %QW."Mag1_AutoWidth".Controlword_6040;
	::MagAWOpen1:tyParamInDriver.uiStatword_6041 AT %IW."Mag1_AutoWidth".Statusword_6041;
	::MagAWOpen1:tyParamOutDriver.siModOfOpt_6060 AT %QB."Mag1_AutoWidth".ModesOfOperation_6060;
	::MagAWOpen1:tyParamInDriver.siModOfOptDisp_6061 AT %IB."Mag1_AutoWidth".ModesOfOperationDisplay_6061;
	::MagAWOpen1:tyParamInDriver.diActualPos_6064 AT %ID."Mag1_AutoWidth".PositionActualValue_6064;
	::MagAWOpen1:tyParamOutDriver.diTargetPos_607A AT %QD."Mag1_AutoWidth".TargetPosition_607A;
	::MagAWOpen1:tyParamOutDriver.udiMoveSpd_6081 AT %QD."Mag1_AutoWidth".ProfileVelocity_6081;
	::MagAWOpen1:tyParamOutDriver.siHmMethod_6098 AT %QB."Mag1_AutoWidth".HomingMethod_6098;
	::MagAWOpen1:tyParamInDriver.udiDigitalInputs_60FD AT %ID."Mag1_AutoWidth".DigitalInputs_60FD;
	::MagAWOpen1:tyParamOutDriver.diJogVel_60FF AT %QD."Mag1_AutoWidth".TargetVelocity_60FF;
	::MagAWOpen2:bModuleOK AT %IX."Mag2_AutoWidth".ModuleOk;
	::MagAWOpen2:tyParamInDriver.uiErrCode_603F AT %IW."Mag2_AutoWidth".ErrorCode_603F;
	::MagAWOpen2:tyParamOutDriver.uiCtrlword_6040 AT %QW."Mag2_AutoWidth".Controlword_6040;
	::MagAWOpen2:tyParamInDriver.uiStatword_6041 AT %IW."Mag2_AutoWidth".Statusword_6041;
	::MagAWOpen2:tyParamOutDriver.siModOfOpt_6060 AT %QB."Mag2_AutoWidth".ModesOfOperation_6060;
	::MagAWOpen2:tyParamInDriver.siModOfOptDisp_6061 AT %IB."Mag2_AutoWidth".ModesOfOperationDisplay_6061;
	::MagAWOpen2:tyParamInDriver.diActualPos_6064 AT %ID."Mag2_AutoWidth".PositionActualValue_6064;
	::MagAWOpen2:tyParamOutDriver.diTargetPos_607A AT %QD."Mag2_AutoWidth".TargetPosition_607A;
	::MagAWOpen2:tyParamOutDriver.udiMoveSpd_6081 AT %QD."Mag2_AutoWidth".ProfileVelocity_6081;
	::MagAWOpen2:tyParamOutDriver.siHmMethod_6098 AT %QB."Mag2_AutoWidth".HomingMethod_6098;
	::MagAWOpen2:tyParamInDriver.udiDigitalInputs_60FD AT %ID."Mag2_AutoWidth".DigitalInputs_60FD;
	::MagAWOpen2:tyParamOutDriver.diJogVel_60FF AT %QD."Mag2_AutoWidth".TargetVelocity_60FF;
	::MagAWOpen3:bModuleOK AT %IX."Mag3_AutoWidth".ModuleOk;
	::MagAWOpen3:tyParamInDriver.uiErrCode_603F AT %IW."Mag3_AutoWidth".ErrorCode_603F;
	::MagAWOpen3:tyParamOutDriver.uiCtrlword_6040 AT %QW."Mag3_AutoWidth".Controlword_6040;
	::MagAWOpen3:tyParamInDriver.uiStatword_6041 AT %IW."Mag3_AutoWidth".Statusword_6041;
	::MagAWOpen3:tyParamOutDriver.siModOfOpt_6060 AT %QB."Mag3_AutoWidth".ModesOfOperation_6060;
	::MagAWOpen3:tyParamInDriver.siModOfOptDisp_6061 AT %IB."Mag3_AutoWidth".ModesOfOperationDisplay_6061;
	::MagAWOpen3:tyParamInDriver.diActualPos_6064 AT %ID."Mag3_AutoWidth".PositionActualValue_6064;
	::MagAWOpen3:tyParamOutDriver.diTargetPos_607A AT %QD."Mag3_AutoWidth".TargetPosition_607A;
	::MagAWOpen3:tyParamOutDriver.udiMoveSpd_6081 AT %QD."Mag3_AutoWidth".ProfileVelocity_6081;
	::MagAWOpen3:tyParamOutDriver.siHmMethod_6098 AT %QB."Mag3_AutoWidth".HomingMethod_6098;
	::MagAWOpen3:tyParamInDriver.udiDigitalInputs_60FD AT %ID."Mag3_AutoWidth".DigitalInputs_60FD;
	::MagAWOpen3:tyParamOutDriver.diJogVel_60FF AT %QD."Mag3_AutoWidth".TargetVelocity_60FF;
	::DOutput:a_bPhysicalDO[43] AT %QX."X20DO9321c".DigitalOutput01;
	::DOutput:a_bPhysicalDO[44] AT %QX."X20DO9321c".DigitalOutput02;
	::DOutput:a_bPhysicalDO[45] AT %QX."X20DO9321c".DigitalOutput03;
	::DOutput:a_bPhysicalDO[46] AT %QX."X20DO9321c".DigitalOutput04;
	::DOutput:a_bPhysicalDO[47] AT %QX."X20DO9321c".DigitalOutput05;
	::DOutput:a_bPhysicalDO[48] AT %QX."X20DO9321c".DigitalOutput06;
	::DOutput:a_bPhysicalDO[49] AT %QX."X20DO9321c".DigitalOutput07;
	::DOutput:a_bPhysicalDO[50] AT %QX."X20DO9321c".DigitalOutput08;
	::DOutput:a_bPhysicalDO[51] AT %QX."X20DO9321c".DigitalOutput09;
	::DOutput:a_bPhysicalDO[52] AT %QX."X20DO9321c".DigitalOutput10;
	::DOutput:a_bPhysicalDO[53] AT %QX."X20DO9321c".DigitalOutput11;
	::DOutput:a_bPhysicalDO[54] AT %QX."X20DO9321c".DigitalOutput12;
	::AWPushOrPu:bModuleOK AT %IX."AutoWidthPusher".ModuleOk;
	::AWPushOrPu:tyParamInDriver.uiErrCode_603F AT %IW."AutoWidthPusher".ErrorCode_603F;
	::AWPushOrPu:tyParamInDriver.uiStatword_6041 AT %IW."AutoWidthPusher".Statusword_6041;
	::AWPushOrPu:tyParamInDriver.siModOfOptDisp_6061 AT %IB."AutoWidthPusher".ModesOfOperationDisplay_6061;
	::AWPushOrPu:tyParamInDriver.diActualPos_6064 AT %ID."AutoWidthPusher".PositionActualValue_6064;
	::AWPushOrPu:tyParamInDriver.udiDigitalInputs_60FD AT %ID."AutoWidthPusher".DigitalInputs_60FD;
	::AWPushOrPu:tyParamOutDriver.uiCtrlword_6040 AT %QW."AutoWidthPusher".Controlword_6040;
	::AWPushOrPu:tyParamOutDriver.siModOfOpt_6060 AT %QB."AutoWidthPusher".ModesOfOperation_6060;
	::AWPushOrPu:tyParamOutDriver.diTargetPos_607A AT %QD."AutoWidthPusher".TargetPosition_607A;
	::AWPushOrPu:tyParamOutDriver.udiMoveSpd_6081 AT %QD."AutoWidthPusher".ProfileVelocity_6081;
	::AWPushOrPu:tyParamOutDriver.siHmMethod_6098 AT %QB."AutoWidthPusher".HomingMethod_6098;
	::AWPushOrPu:tyParamOutDriver.diJogVel_60FF AT %QD."AutoWidthPusher".TargetVelocity_60FF;
	::AWPushOrPu:tyParamOutDriver.siModOfOpt_6060 AT %QB."AutoWidthPusher".Modes_of_operation_6060;
	::AWPushOrPu:tyParamOutDriver.diTargetPos_607A AT %QD."AutoWidthPusher".Target_position_607A;
	::AWPushOrPu:tyParamOutDriver.udiMoveSpd_6081 AT %QD."AutoWidthPusher".Profile_velocity_6081;
	::AWPushOrPu:tyParamOutDriver.siHmMethod_6098 AT %QB."AutoWidthPusher".Homing_method_6098;
	::AWPushOrPu:tyParamOutDriver.diJogVel_60FF AT %QD."AutoWidthPusher".Target_velocity_60FF;
	::AWPushOrPu:tyParamInDriver.uiErrCode_603F AT %IW."AutoWidthPusher".Error_code_603F;
	::AWPushOrPu:tyParamInDriver.siModOfOptDisp_6061 AT %IB."AutoWidthPusher".Modes_of_operation_display_6061;
	::AWPushOrPu:tyParamInDriver.diActualPos_6064 AT %ID."AutoWidthPusher".Position_actual_value_6064;
	::AWPushOrPu:tyParamInDriver.udiDigitalInputs_60FD AT %ID."AutoWidthPusher".Digital_intputs_60FD;
	::PullerPush:bModuleOK AT %IX."PullerPusher".ModuleOk;
	::PullerPush:tyParamInDriver.uiErrCode_603F AT %IW."PullerPusher".ErrorCode_603F;
	::PullerPush:tyParamInDriver.uiStatword_6041 AT %IW."PullerPusher".Statusword_6041;
	::PullerPush:tyParamInDriver.siModOfOptDisp_6061 AT %IB."PullerPusher".ModesOfOperationDisplay_6061;
	::PullerPush:tyParamInDriver.udiDigitalInputs_60FD AT %ID."PullerPusher".DigitalInputs_60FD;
	::PullerPush:tyParamOutDriver.uiCtrlword_6040 AT %QW."PullerPusher".Controlword_6040;
	::PullerPush:tyParamOutDriver.siModOfOpt_6060 AT %QB."PullerPusher".ModesOfOperation_6060;
	::PullerPush:tyParamInDriver.diActualPos_6064 AT %ID."PullerPusher".PositionActualValue_6064;
	::PullerPush:tyParamOutDriver.diTargetPos_607A AT %QD."PullerPusher".TargetPosition_607A;
	::PullerPush:tyParamOutDriver.udiMoveSpd_6081 AT %QD."PullerPusher".ProfileVelocity_6081;
	::PullerPush:tyParamOutDriver.siHmMethod_6098 AT %QB."PullerPusher".HomingMethod_6098;
	::PullerPush:tyParamOutDriver.diJogVel_60FF AT %QD."PullerPusher".TargetVelocity_60FF;
END_VAR
```

### Acp10cfg.ncc - X20CP0483/Motion/Acp10cfg.ncc
```
NcConfiguration (Version=5.08.2, NcSwId=Acp10)
  ACP10CF1_typ:
    cnt_nettrc_rec_drive = 150
    bufsize_trace_upload = 1200
    tc_nc_man_task = Cyclic #1
    glob_pv_as_ncobject = Yes
    ncsys_dl_broadcast = Yes
    ncsys_dl_acp_reset = Yes
    safemc_log_err_to_ax = Yes
    network_init:
      ncsw_init_execute = Yes
      automatic_execute = No
      node_nr_warning = Yes
      net_err_before_ncact = Yes
    nettrc:
      enter_parsecrec = Yes
      enter_ncaction = Yes
      save_ring_startidx = No
    cam_prof_download:
      cam_dat_dl_parallel = No
      tc_cam_dl_parallel = Task class for NC Manager task
```

## Configuration 3Mag_UL_MagPlat

### Task classes (Cpu.sw)
```
Cyclic#1 (cycle 10000 us, tolerance 10000 us):
  DInput <- DInput.DInput.prg
  DOutput <- DOutput.DOutput.prg
  PneuNoSen8 <- (binary)
  PneuNoSen4 <- (binary)
  PneuNoSenT <- (binary)
  PneuNoSen9 <- (binary)
  PneuNoSenB <- (binary)
  PneuNoSen7 <- (binary)
  Lifter2 <- (binary)
  PneuNoSe10 <- (binary)
  PneuNoSen3 <- (binary)
  PneuNoSen6 <- (binary)
  PneuNoSen5 <- (binary)
  InMagConv <- (binary)
  LifterMag1 <- (binary)
  LifterMagC <- (binary)
  OutMagConv <- (binary)
  OutMagCon1 <- (binary)
  OpCon <- (binary)
  InMagConv2 <- (binary)
  TCP1 <- (binary)
  TCP <- (binary)
  TCP2 <- (binary)
Cyclic#2 (cycle 20000 us, tolerance 20000 us):
  PshrConv <- Conv.PshrConv.prg
  MtrPshr <- MtrPshr.MtrPshr.prg
  PullerPush <- CANOpenServo.PullerPusher.PullerPusher.prg
  MagConv2Cl <- MagConv_LiftnTrav.MagConv2Clp1.prg
  MagConv2C1 <- MagConv_LiftnTrav.MagConv2Clp2.prg
  MagConv2C2 <- MagConv_LiftnTrav.MagConv2Clp3.prg
Cyclic#3 (cycle 50000 us, tolerance 50000 us):
  UI <- UI.UI.prg
  Startup <- Startup.Startup.prg
  General <- General.General.prg
  UsrFolder <- UsrFolder.UsrFolder.prg
  LibVer <- LibVer.LibVer.prg
  HWInfo <- HWInfo.HWInfo.prg
  Alarm <- Alarm.Alarm.prg
  TLBuz <- TLBuz.TLBuz.prg
  ProdRcp <- ProdRcp.ProdRcp.prg
  MpProdRcp <- MpProdRcp.MpProdRcp.prg
  MagRcp <- MagRcp.MagRcp.prg
  McParam <- McParam.McParam.prg
  NtParam <- NtParam.NtParam.prg
  UsrMgmt <- UsrMgmt.UsrMgmt.prg
  OvenInfoA <- OvenInfo.OvenInfoA.prg
  OvenInfoB <- OvenInfo.OvenInfoB.prg
  Buffer1 <- Buffer.Buffer1.prg
  Buffer2 <- Buffer.Buffer2.prg
  Buffer3 <- Buffer.Buffer3.prg
  BufferMagA <- Buffer.BufferMagA.prg
  BufferMagB <- Buffer.BufferMagB.prg
  USSMEMAA <- SMEMA.USSMEMAA.prg
  USSMEMAB <- SMEMA.USSMEMAB.prg
  USSMEMA1 <- SMEMA.USSMEMA1.prg
  USSMEMA2 <- SMEMA.USSMEMA2.prg
  USSMEMA3 <- SMEMA.USSMEMA3.prg
  DSSMEMA1 <- SMEMA.DSSMEMA1.prg
  DSSMEMA2 <- SMEMA.DSSMEMA2.prg
  DSSMEMA3 <- SMEMA.DSSMEMA3.prg
  Pneu2SenIn <- Pneu.PneuInShutter.prg
  Pneu2SenOu <- Pneu.PneuOutShutter.prg
  Pneu2SenO1 <- Pneu.PneuOutShutter2.prg
  Pneu2SenO2 <- Pneu.PneuOutShutter3.prg
  PneuNoSenS <- Pneu.PneuStopperA.prg
  PneuNoSen1 <- Pneu.PneuStopperB.prg
  PneuNoSen2 <- Pneu.PneuStopperC.prg
  Pneu2SenSe <- Pneu.PneuSelClamp1.prg
  Pneu2SenMa <- Pneu.PneuMag1SafetyBar.prg
  Pneu2SenM3 <- Pneu.PneuMag1AWEngage.prg
  Trav <- CANOpenServo.Trav.Trav.prg
  LifterBtm <- CANOpenServo.Lifter.LifterBtm.prg
  MagAWOpen1 <- CANOpenServo.MagAW.MagAWOpen1.prg
  MagAWOpen2 <- CANOpenServo.MagAW.MagAWOpen2.prg
  MagAWOpen3 <- CANOpenServo.MagAW.MagAWOpen3.prg
  Hermes <- Hermes.Hermes.prg
  USHermesA <- Hermes.USHermesA.prg
  USHermesB <- Hermes.USHermesB.prg
  RmtHermes <- Hermes.RmtHermes.prg
  SvyHermes <- Hermes.SvyHermes.prg
  LCS <- LCS.LCS.prg
  LCSMngRcp <- LCS.LCSMngRcp.prg
  LCSLF <- LCS.LCSLF.prg
  LFLeader <- LF.LFLeader.prg
  LFFollower <- LF.LFFollower.prg
  Follower1 <- LF.Follower1.prg
  Follower2 <- LF.Follower2.prg
  AWOpen <- CANOpenServo.AW.AWOpen.prg
  AWPushOrPu <- CANOpenServo.AW.AWPushOrPuller.prg
  Ops <- Operations.Ops.prg
  OpsTravLif <- Operations.OpsTravLifUL.prg
  OpsMagConv <- Operations.MagConv_StationaryPlat.OpsMagConvUL1.prg
  OpsMagCon1 <- Operations.MagConv_StationaryPlat.OpsMagConvUL2.prg
  OpsMagCon2 <- Operations.MagConv_StationaryPlat.OpsMagConvUL3.prg
  OpsLifMagU <- Operations.OpsLifMagUL.prg
  AGV <- AGVCom.AGV.prg
  AGV1 <- AGVCom.AGV1.prg
  AGV2 <- AGVCom.AGV2.prg
  AGV3 <- AGVCom.AGV3.prg
  Simu <- Simulation.Simu.prg
  AutoRcp <- AutoRcp.AutoRcp.prg
  Machine <- Machine.Machine.prg
  USSOT1 <- SOT.USSOT1.prg
  DSSOT1 <- SOT.DSSOT1.prg
  USSOT2 <- SOT.USSOT2.prg
  DSSOT2 <- SOT.DSSOT2.prg
  USSOT3 <- SOT.USSOT3.prg
  DSSOT3 <- SOT.DSSOT3.prg
  Simu1 <- Simulation.Simu1.prg
Cyclic#4 (cycle 10000 us, tolerance 10000 us):
  RstErr <- RstErr.RstErr.prg
DataObjects: Acp10sys
VcDataObjects: Visu <- UI.Visu.dob
Binaries: vcfntttf, arialbi, vccbmp, vcshared, vcpdvnc, vccshape, vcfile, vcgclass, arial, vcchspot, vcmgr, arialxsr, vccslider, vcdsint, vccbtn, vcdsloc, vccovl, vccpopup, vccline, vcctext, vcalarm, vcbclass, vccbar, visvc, udbdef, vcrt, vccnum, vccstr, Visu03, vccddbox, arialbd, vcpdsw, vcnet, TCData, Visu02, Visu01, vctcal, vccdt, vccalarm, arsvcreg, vcpfgen, acp10cfg, Acp10map, arconfig, asfw, iomap, Role, ashwd, ashwac, sysconf, User, Config, vcpfar00, OpcUaMap
Libraries: standard, runtime, astime, asstring, operator, AsIecCon, AsCANopen, visapi, FileIO, AsIODiag, AsMem, dvframe, AsOpcUac, AsARCfg, sys_lib, AsTCP, AsFltGen, brsystem, MpCom, MpBase, MpRecipe, Acp10man, Acp10par, NcGlobal, AsMath, NtBuffer, NtConv, NtFileIO, NtLogFile, NtMem, NtMessage, NtOvenInfo, NtPneu, NtRS232, NtSMEMA, NtTCP, NtTLBuz, NtVersion, NtSOT, NtLF, NtMotion, NtRecipe, NtGeneral, NtUI, NtHermes, NtOpConXML, NtOPCUA, dataobj, vcresman, powerlnk
```

### Hardware
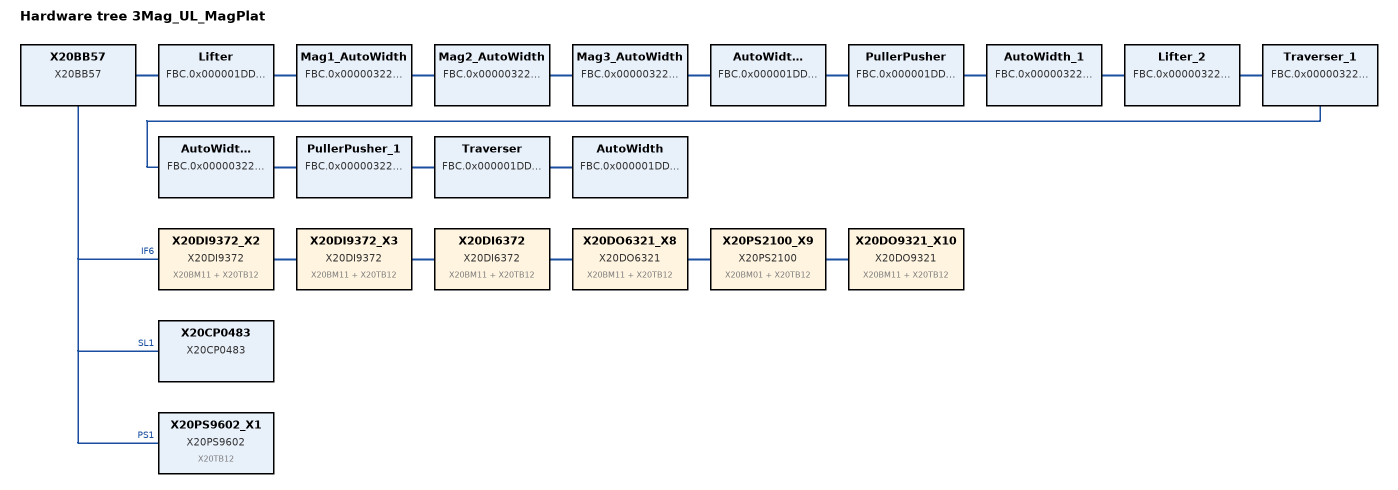
```
AutoWidth : FBC.0x000001DD.0x00000001.NUTEK_DELTA_EDS_V101 v1.0 (OrderNumber=NUTEK_DELTA_V101)  [CAN1 -> Traverser.CAN2 (NodeNumber=16)]
AutoWidthPusher : FBC.0x000001DD.0x00000001.NUTEK_DELTA_EDS_V101 v1.0 (OrderNumber=NUTEK_DELTA_V101)  [CAN1 -> Mag3_AutoWidth.CAN2]
AutoWidthPusher_1 : FBC.0x00000322.0x00001000.NUTEK_ESTUN_PronetPlus_EDS_V106 v1.06.1 (Disabled=true, OrderNumber=NUTEK_ESTUN_PronetPlus_V106)  [CAN1 -> Traverser_1.CAN2]
AutoWidth_1 : FBC.0x00000322.0x00001000.NUTEK_ESTUN_PronetPlus_EDS_V106 v1.06.1 (Disabled=true, OrderNumber=NUTEK_ESTUN_PronetPlus_V106)  [CAN1 -> PullerPusher.CAN2]
Lifter : FBC.0x000001DD.0x00000001.NUTEK_DELTA_EDS_V101 v1.0 (OrderNumber=NUTEK_DELTA_V101)  [CAN1 -> X20BB57.IF7 (NodeNumber=17)]
Lifter_2 : FBC.0x00000322.0x00001000.NUTEK_ESTUN_PronetPlus_EDS_V106 v1.06.1 (Disabled=true, OrderNumber=NUTEK_ESTUN_PronetPlus_V106)  [CAN1 -> AutoWidth_1.CAN2]
Mag1_AutoWidth : FBC.0x00000322.0x00001000.NUTEK_ESTUN_PronetPlus_EDS_V106 v1.06.1 (Disabled=true, OrderNumber=NUTEK_ESTUN_PronetPlus_V106)  [CAN1 -> Lifter.CAN2 (NodeNumber=19)]
Mag2_AutoWidth : FBC.0x00000322.0x00001000.NUTEK_ESTUN_PronetPlus_EDS_V106 v1.06.1 (Disabled=true, OrderNumber=NUTEK_ESTUN_PronetPlus_V106)  [CAN1 -> Mag1_AutoWidth.CAN2]
Mag3_AutoWidth : FBC.0x00000322.0x00001000.NUTEK_ESTUN_PronetPlus_EDS_V106 v1.06.1 (Disabled=true, OrderNumber=NUTEK_ESTUN_PronetPlus_V106)  [CAN1 -> Mag2_AutoWidth.CAN2]
PullerPusher : FBC.0x000001DD.0x00000001.NUTEK_DELTA_EDS_V101 v1.0 (OrderNumber=NUTEK_DELTA_V101)  [CAN1 -> AutoWidthPusher.CAN2]
PullerPusher_1 : FBC.0x00000322.0x00001000.NUTEK_ESTUN_PronetPlus_EDS_V106 v1.06.1 (Disabled=true, OrderNumber=NUTEK_ESTUN_PronetPlus_V106)  [CAN1 -> AutoWidthPusher_1.CAN2]
Traverser : FBC.0x000001DD.0x00000001.NUTEK_DELTA_EDS_V101 v1.0 (OrderNumber=NUTEK_DELTA_V101)  [CAN1 -> PullerPusher_1.CAN2 (NodeNumber=18)]
Traverser_1 : FBC.0x00000322.0x00001000.NUTEK_ESTUN_PronetPlus_EDS_V106 v1.06.1 (Disabled=true, OrderNumber=NUTEK_ESTUN_PronetPlus_V106)  [CAN1 -> Lifter_2.CAN2]
X20BB57 : X20BB57 v1.1.1.0
  Connector IF1:
    Baudrate = 9600
    Parity = N
  Connector IF7:
    Baudrate = 1000000
    ActivateCanOpen = 1
    p100c_parametervalue = 1000
    p100d_parametervalue = 3
X20BM01 : X20BM01 v2.1.0.0  [X2X1 -> X20BM11e.X2X2]
X20BM11 : X20BM11 v1.0.0.1  [X2X1 -> X20BB57.IF6]
X20BM11a : X20BM11 v1.0.0.1  [X2X1 -> X20BM11.X2X2]
X20BM11b : X20BM11 v1.0.0.1  [X2X1 -> X20BM11a.X2X2]
X20BM11e : X20BM11 v1.0.0.1  [X2X1 -> X20BM11b.X2X2]
X20BM11f : X20BM11 v1.0.0.1  [X2X1 -> X20BM01.X2X2]
X20CP0483 : X20CP0483 v1.2.1.0  [SL -> X20BB57.SL1]
  Connector IF2:
    ActivateDevice = 1
    Mode = Manual
    InternetAddress = 192.168.0.10
    SubnetMask = 255.255.255.0
    InaNodeNumber = 36
    Vnc1
    VncVcObjectName1 = Visu
    VncKeyMappingFile1 = 
    VncMaxConnections1 = 3
    VncRefreshRate1 = 100
    ActivateSnmp = 2
  Connector IF3:
    Operation = EthOnly
    EthernetMode = Manual
    InternetAddress = 192.168.2.100
    SubnetMask = 255.255.255.0
    ActivateSnmp = 2
  ConfigurationID = NAEUL004
  UserPartitionSize = 150
  VolatileGlobalPvSize = 50000
  EnableUsbRemoteInstall = 1
  TimerDeviceType = SWIOTIMER
  Cyclic1Duration = 10000
  Cyclic1Tolerance = 10000
  Cyclic2Duration = 20000
  Cyclic2Tolerance = 20000
  Cyclic3Duration = 50000
  Cyclic3Tolerance = 50000
  Cyclic4Duration = 10000
  Cyclic4Tolerance = 10000
  Cyclic5Duration = 200000
  Cyclic5Tolerance = 200000
  Cyclic6Duration = 500000
  Cyclic6Tolerance = 500000
  Cyclic7Duration = 1000000
  Cyclic7Tolerance = 1000000
  Cyclic8Duration = 10000
  Cyclic8Tolerance = 10000
  FileDevice1
  FileDeviceName1 = F
  FileDevicePath1 = F:
  FileDevice2
  FileDeviceName2 = User
  FileDevicePath2 = F:\User
  FileDevice3
  FileDeviceName3 = Private
  FileDevicePath3 = F:\Private
  FileDevice4
  FileDeviceName4 = CustomerUser
  FileDevicePath4 = F:\User\UserMgmt
  FileDevice5
  FileDeviceName5 = ProdRcp
  FileDevicePath5 = F:\User\ProductRecipe
  FileDevice6
  FileDeviceName6 = MagRcp
  FileDevicePath6 = F:\User\MagazineRecipe
  FileDevice7
  FileDeviceName7 = Alarm
  FileDevicePath7 = F:\User\Alarm
  FileDevice8
  FileDeviceName8 = McParam
  FileDevicePath8 = F:\User\MachineParameter
  FileDevice9
  FileDeviceName9 = NtParam
  FileDevicePath9 = F:\Private\NutekParameter
  FileDevice10
  FileDeviceName10 = LibVer
  FileDevicePath10 = F:\User\LibrariesVersion
  FileDevice11
  FileDeviceName11 = Retain
  FileDevicePath11 = F:\User\Retain
  FileDevice12
  FileDeviceName12 = Log
  FileDevicePath12 = F:\User\Log
  FileDevice13
  FileDeviceName13 = LCS
  FileDevicePath13 = F:\User\LCS
  FileDevice14
  FileDeviceName14 = MpProdRcp
  FileDevicePath14 = F:\User\ProductRecipeXml
  FileDevice15
  FileDeviceName15 = MpNtParam
  FileDevicePath15 = F:\Private\NutekParameterXml
  FtpUser1
  FtpUsername1 = NTAFTP
  FtpUserPassword1 = +UZ5u8Axw7KkkY4oM/r7wOOfB5oWHxpSY6r3j++jJso=  // NTA4BH
  FtpUserSalt1 = c0Alfi1W
  FTPAccessRight1 = 0
  FTPdevice1 = ALL
  FtpUser2
  FtpUsername2 = admin
  FtpUserPassword2 = mW+qRsE1LOSFDAB60rBJwb9dZ7uQUIuoHZp04C+x5XU=  // admin
  FtpUserSalt2 = Nr9+IHjr
  FTPAccessRight2 = 0
  FTPMSpath2 = User
  FtpUser3
  FtpUsername3 = LCS
  FtpUserPassword3 = W4lkF6NjcyaB1sRdLwIoSAlqHoAE4GimWQdq7pKTzbA=  // LCS
  FtpUserSalt3 = f3H7b7h0
  FTPMSpath3 = User\LCS
  FtpUser4
  FtpUsername4 = user
  FtpUserPassword4 = aIGm/evksyHJRue4841xDUns9BsVPAD8aaNpA7aBGks=  // user
  FtpUserSalt4 = o5eEPKTD
  FTPMSpath4 = User\ProductRecipeXml
  ActivateOpcUa = 1
  OpcUa_ConversationSecurityPolicy_EnableBasic256Rsa256 = 0
  OpcUaInformationModels_PV_Version = 1
X20DI6372 : X20DI6372 v1.1.0.0  [SS1 -> X20TB12c.SS; SL -> X20BM11b.SL1]
X20DI9372_X2 : X20DI9372 v1.1.0.0  [SS1 -> X20TB12a.SS; SL -> X20BM11.SL1]
X20DI9372_X3 : X20DI9372 v1.1.0.0  [SS1 -> X20TB12b.SS; SL -> X20BM11a.SL1]
X20DO6321_X8 : X20DO6321 v1.1.0.0  [SS1 -> X20TB12f.SS; SL -> X20BM11e.SL1]
X20DO9321_X10 : X20DO9321 v1.1.0.0  [SS1 -> X20TB12h.SS; SL -> X20BM11f.SL1]
X20PS2100_X9 : X20PS2100 v1.2.0.0  [SS1 -> X20TB12g.SS; SL -> X20BM01.SL1]
X20PS9602_X1 : X20PS9602 v1.0.2.0  [PS -> X20BB57.PS1; SS1 -> X20TB12.SS]
X20TB12 : X20TB12 v1.0.0.0
X20TB12a : X20TB12 v1.0.0.0
X20TB12b : X20TB12 v1.0.0.0
X20TB12c : X20TB12 v1.0.0.0
X20TB12f : X20TB12 v1.0.0.0
X20TB12g : X20TB12 v1.0.0.0
X20TB12h : X20TB12 v1.0.0.0
```

### IoMap.iom - X20CP0483/IoMap.iom
```iecst
VAR_CONFIG
	::AWOpen:bModuleOK AT %IX."AutoWidth".ModuleOk;
	::AWOpen:tyParamInDriver.uiErrCode_603F AT %IW."AutoWidth".ErrorCode_603F;
	::AWOpen:tyParamOutDriver.uiCtrlword_6040 AT %QW."AutoWidth".Controlword_6040;
	::AWOpen:tyParamInDriver.uiStatword_6041 AT %IW."AutoWidth".Statusword_6041;
	::AWOpen:tyParamOutDriver.siModOfOpt_6060 AT %QB."AutoWidth".ModesOfOperation_6060;
	::AWOpen:tyParamInDriver.siModOfOptDisp_6061 AT %IB."AutoWidth".ModesOfOperationDisplay_6061;
	::AWOpen:tyParamInDriver.diActualPos_6064 AT %ID."AutoWidth".PositionActualValue_6064;
	::AWOpen:tyParamOutDriver.diTargetPos_607A AT %QD."AutoWidth".TargetPosition_607A;
	::AWOpen:tyParamOutDriver.udiMoveSpd_6081 AT %QD."AutoWidth".ProfileVelocity_6081;
	::AWOpen:tyParamOutDriver.siHmMethod_6098 AT %QB."AutoWidth".HomingMethod_6098;
	::AWOpen:tyParamInDriver.udiDigitalInputs_60FD AT %ID."AutoWidth".DigitalInputs_60FD;
	::AWOpen:tyParamOutDriver.diJogVel_60FF AT %QD."AutoWidth".TargetVelocity_60FF;
	::LifterBtm:bModuleOK AT %IX."Lifter".ModuleOk;
	::LifterBtm:tyParamInDriver.uiErrCode_603F AT %IW."Lifter".ErrorCode_603F;
	::LifterBtm:tyParamOutDriver.uiCtrlword_6040 AT %QW."Lifter".Controlword_6040;
	::LifterBtm:tyParamInDriver.uiStatword_6041 AT %IW."Lifter".Statusword_6041;
	::LifterBtm:tyParamOutDriver.siModOfOpt_6060 AT %QB."Lifter".ModesOfOperation_6060;
	::LifterBtm:tyParamInDriver.siModOfOptDisp_6061 AT %IB."Lifter".ModesOfOperationDisplay_6061;
	::LifterBtm:tyParamInDriver.diActualPos_6064 AT %ID."Lifter".PositionActualValue_6064;
	::LifterBtm:tyParamOutDriver.diTargetPos_607A AT %QD."Lifter".TargetPosition_607A;
	::LifterBtm:tyParamOutDriver.udiMoveSpd_6081 AT %QD."Lifter".ProfileVelocity_6081;
	::LifterBtm:tyParamOutDriver.siHmMethod_6098 AT %QB."Lifter".HomingMethod_6098;
	::LifterBtm:tyParamInDriver.udiDigitalInputs_60FD AT %ID."Lifter".DigitalInputs_60FD;
	::LifterBtm:tyParamOutDriver.diJogVel_60FF AT %QD."Lifter".TargetVelocity_60FF;
	::DInput:a_bPhysicalDI[1] AT %IX."X20DI9372_X2".DigitalInput01;
	::DInput:a_bPhysicalDI[2] AT %IX."X20DI9372_X2".DigitalInput02;
	::DInput:a_bPhysicalDI[3] AT %IX."X20DI9372_X2".DigitalInput03;
	::DInput:a_bPhysicalDI[4] AT %IX."X20DI9372_X2".DigitalInput04;
	::DInput:a_bPhysicalDI[5] AT %IX."X20DI9372_X2".DigitalInput05;
	::DInput:a_bPhysicalDI[6] AT %IX."X20DI9372_X2".DigitalInput06;
	::DInput:a_bPhysicalDI[7] AT %IX."X20DI9372_X2".DigitalInput07;
	::DInput:a_bPhysicalDI[8] AT %IX."X20DI9372_X2".DigitalInput08;
	::DInput:a_bPhysicalDI[9] AT %IX."X20DI9372_X2".DigitalInput09;
	::DInput:a_bPhysicalDI[10] AT %IX."X20DI9372_X2".DigitalInput10;
	::DInput:a_bPhysicalDI[11] AT %IX."X20DI9372_X2".DigitalInput11;
	::DInput:a_bPhysicalDI[12] AT %IX."X20DI9372_X2".DigitalInput12;
	::DInput:a_bPhysicalDI[13] AT %IX."X20DI9372_X3".DigitalInput01;
	::DInput:a_bPhysicalDI[14] AT %IX."X20DI9372_X3".DigitalInput02;
	::DInput:a_bPhysicalDI[15] AT %IX."X20DI9372_X3".DigitalInput03;
	::DInput:a_bPhysicalDI[16] AT %IX."X20DI9372_X3".DigitalInput04;
	::DInput:a_bPhysicalDI[17] AT %IX."X20DI9372_X3".DigitalInput05;
	::DInput:a_bPhysicalDI[18] AT %IX."X20DI9372_X3".DigitalInput06;
	::DInput:a_bPhysicalDI[19] AT %IX."X20DI9372_X3".DigitalInput07;
	::DInput:a_bPhysicalDI[20] AT %IX."X20DI9372_X3".DigitalInput08;
	::DInput:a_bPhysicalDI[21] AT %IX."X20DI9372_X3".DigitalInput09;
	::DInput:a_bPhysicalDI[22] AT %IX."X20DI9372_X3".DigitalInput10;
	::DInput:a_bPhysicalDI[23] AT %IX."X20DI9372_X3".DigitalInput11;
	::DInput:a_bPhysicalDI[24] AT %IX."X20DI9372_X3".DigitalInput12;
	::DInput:a_bPhysicalDI[25] AT %IX."X20DI6372".DigitalInput01;
	::DInput:a_bPhysicalDI[26] AT %IX."X20DI6372".DigitalInput02;
	::DInput:a_bPhysicalDI[27] AT %IX."X20DI6372".DigitalInput03;
	::DInput:a_bPhysicalDI[28] AT %IX."X20DI6372".DigitalInput04;
	::DInput:a_bPhysicalDI[29] AT %IX."X20DI6372".DigitalInput05;
	::DInput:a_bPhysicalDI[30] AT %IX."X20DI6372".DigitalInput06;
	::DOutput:a_bPhysicalDO[1] AT %QX."X20DO6321_X8".DigitalOutput01;
	::DOutput:a_bPhysicalDO[2] AT %QX."X20DO6321_X8".DigitalOutput02;
	::DOutput:a_bPhysicalDO[3] AT %QX."X20DO6321_X8".DigitalOutput03;
	::DOutput:a_bPhysicalDO[4] AT %QX."X20DO6321_X8".DigitalOutput04;
	::DOutput:a_bPhysicalDO[5] AT %QX."X20DO6321_X8".DigitalOutput05;
	::DOutput:a_bPhysicalDO[6] AT %QX."X20DO6321_X8".DigitalOutput06;
	::DOutput:a_bPhysicalDO[7] AT %QX."X20DO9321_X10".DigitalOutput01;
	::DOutput:a_bPhysicalDO[8] AT %QX."X20DO9321_X10".DigitalOutput02;
	::DOutput:a_bPhysicalDO[9] AT %QX."X20DO9321_X10".DigitalOutput03;
	::DOutput:a_bPhysicalDO[10] AT %QX."X20DO9321_X10".DigitalOutput04;
	::DOutput:a_bPhysicalDO[11] AT %QX."X20DO9321_X10".DigitalOutput05;
	::DOutput:a_bPhysicalDO[12] AT %QX."X20DO9321_X10".DigitalOutput06;
	::DOutput:a_bPhysicalDO[13] AT %QX."X20DO9321_X10".DigitalOutput07;
	::DOutput:a_bPhysicalDO[14] AT %QX."X20DO9321_X10".DigitalOutput08;
	::DOutput:a_bPhysicalDO[15] AT %QX."X20DO9321_X10".DigitalOutput09;
	::DOutput:a_bPhysicalDO[16] AT %QX."X20DO9321_X10".DigitalOutput10;
	::DOutput:a_bPhysicalDO[17] AT %QX."X20DO9321_X10".DigitalOutput11;
	::DOutput:a_bPhysicalDO[18] AT %QX."X20DO9321_X10".DigitalOutput12;
	::MagAWOpen1:bModuleOK AT %IX."Mag1_AutoWidth".ModuleOk;
	::MagAWOpen1:tyParamInDriver.uiErrCode_603F AT %IW."Mag1_AutoWidth".ErrorCode_603F;
	::MagAWOpen1:tyParamOutDriver.uiCtrlword_6040 AT %QW."Mag1_AutoWidth".Controlword_6040;
	::MagAWOpen1:tyParamInDriver.uiStatword_6041 AT %IW."Mag1_AutoWidth".Statusword_6041;
	::MagAWOpen1:tyParamOutDriver.siModOfOpt_6060 AT %QB."Mag1_AutoWidth".ModesOfOperation_6060;
	::MagAWOpen1:tyParamInDriver.siModOfOptDisp_6061 AT %IB."Mag1_AutoWidth".ModesOfOperationDisplay_6061;
	::MagAWOpen1:tyParamInDriver.diActualPos_6064 AT %ID."Mag1_AutoWidth".PositionActualValue_6064;
	::MagAWOpen1:tyParamOutDriver.diTargetPos_607A AT %QD."Mag1_AutoWidth".TargetPosition_607A;
	::MagAWOpen1:tyParamOutDriver.udiMoveSpd_6081 AT %QD."Mag1_AutoWidth".ProfileVelocity_6081;
	::MagAWOpen1:tyParamOutDriver.siHmMethod_6098 AT %QB."Mag1_AutoWidth".HomingMethod_6098;
	::MagAWOpen1:tyParamInDriver.udiDigitalInputs_60FD AT %ID."Mag1_AutoWidth".DigitalInputs_60FD;
	::MagAWOpen1:tyParamOutDriver.diJogVel_60FF AT %QD."Mag1_AutoWidth".TargetVelocity_60FF;
	::MagAWOpen2:bModuleOK AT %IX."Mag2_AutoWidth".ModuleOk;
	::MagAWOpen2:tyParamInDriver.uiErrCode_603F AT %IW."Mag2_AutoWidth".ErrorCode_603F;
	::MagAWOpen2:tyParamOutDriver.uiCtrlword_6040 AT %QW."Mag2_AutoWidth".Controlword_6040;
	::MagAWOpen2:tyParamInDriver.uiStatword_6041 AT %IW."Mag2_AutoWidth".Statusword_6041;
	::MagAWOpen2:tyParamOutDriver.siModOfOpt_6060 AT %QB."Mag2_AutoWidth".ModesOfOperation_6060;
	::MagAWOpen2:tyParamInDriver.siModOfOptDisp_6061 AT %IB."Mag2_AutoWidth".ModesOfOperationDisplay_6061;
	::MagAWOpen2:tyParamInDriver.diActualPos_6064 AT %ID."Mag2_AutoWidth".PositionActualValue_6064;
	::MagAWOpen2:tyParamOutDriver.diTargetPos_607A AT %QD."Mag2_AutoWidth".TargetPosition_607A;
	::MagAWOpen2:tyParamOutDriver.udiMoveSpd_6081 AT %QD."Mag2_AutoWidth".ProfileVelocity_6081;
	::MagAWOpen2:tyParamOutDriver.siHmMethod_6098 AT %QB."Mag2_AutoWidth".HomingMethod_6098;
	::MagAWOpen2:tyParamInDriver.udiDigitalInputs_60FD AT %ID."Mag2_AutoWidth".DigitalInputs_60FD;
	::MagAWOpen2:tyParamOutDriver.diJogVel_60FF AT %QD."Mag2_AutoWidth".TargetVelocity_60FF;
	::MagAWOpen3:bModuleOK AT %IX."Mag3_AutoWidth".ModuleOk;
	::MagAWOpen3:tyParamInDriver.uiErrCode_603F AT %IW."Mag3_AutoWidth".ErrorCode_603F;
	::MagAWOpen3:tyParamOutDriver.uiCtrlword_6040 AT %QW."Mag3_AutoWidth".Controlword_6040;
	::MagAWOpen3:tyParamInDriver.uiStatword_6041 AT %IW."Mag3_AutoWidth".Statusword_6041;
	::MagAWOpen3:tyParamOutDriver.siModOfOpt_6060 AT %QB."Mag3_AutoWidth".ModesOfOperation_6060;
	::MagAWOpen3:tyParamInDriver.siModOfOptDisp_6061 AT %IB."Mag3_AutoWidth".ModesOfOperationDisplay_6061;
	::MagAWOpen3:tyParamInDriver.diActualPos_6064 AT %ID."Mag3_AutoWidth".PositionActualValue_6064;
	::MagAWOpen3:tyParamOutDriver.diTargetPos_607A AT %QD."Mag3_AutoWidth".TargetPosition_607A;
	::MagAWOpen3:tyParamOutDriver.udiMoveSpd_6081 AT %QD."Mag3_AutoWidth".ProfileVelocity_6081;
	::MagAWOpen3:tyParamOutDriver.siHmMethod_6098 AT %QB."Mag3_AutoWidth".HomingMethod_6098;
	::MagAWOpen3:tyParamInDriver.udiDigitalInputs_60FD AT %ID."Mag3_AutoWidth".DigitalInputs_60FD;
	::MagAWOpen3:tyParamOutDriver.diJogVel_60FF AT %QD."Mag3_AutoWidth".TargetVelocity_60FF;
	::AWPushOrPu:bModuleOK AT %IX."AutoWidthPusher".ModuleOk;
	::AWPushOrPu:tyParamInDriver.uiErrCode_603F AT %IW."AutoWidthPusher".ErrorCode_603F;
	::AWPushOrPu:tyParamInDriver.uiStatword_6041 AT %IW."AutoWidthPusher".Statusword_6041;
	::AWPushOrPu:tyParamInDriver.siModOfOptDisp_6061 AT %IB."AutoWidthPusher".ModesOfOperationDisplay_6061;
	::AWPushOrPu:tyParamInDriver.diActualPos_6064 AT %ID."AutoWidthPusher".PositionActualValue_6064;
	::AWPushOrPu:tyParamInDriver.udiDigitalInputs_60FD AT %ID."AutoWidthPusher".DigitalInputs_60FD;
	::AWPushOrPu:tyParamOutDriver.uiCtrlword_6040 AT %QW."AutoWidthPusher".Controlword_6040;
	::AWPushOrPu:tyParamOutDriver.siModOfOpt_6060 AT %QB."AutoWidthPusher".ModesOfOperation_6060;
	::AWPushOrPu:tyParamOutDriver.diTargetPos_607A AT %QD."AutoWidthPusher".TargetPosition_607A;
	::AWPushOrPu:tyParamOutDriver.udiMoveSpd_6081 AT %QD."AutoWidthPusher".ProfileVelocity_6081;
	::AWPushOrPu:tyParamOutDriver.siHmMethod_6098 AT %QB."AutoWidthPusher".HomingMethod_6098;
	::AWPushOrPu:tyParamOutDriver.diJogVel_60FF AT %QD."AutoWidthPusher".TargetVelocity_60FF;
	::AWOpen:tyParamInDriver.uiErrCode_603F AT %IW."AutoWidth".Error_code_603F;
	::AWOpen:tyParamInDriver.siModOfOptDisp_6061 AT %IB."AutoWidth".Modes_of_operation_display_6061;
	::AWOpen:tyParamInDriver.diActualPos_6064 AT %ID."AutoWidth".Position_actual_value_6064;
	::AWOpen:tyParamInDriver.udiDigitalInputs_60FD AT %ID."AutoWidth".Digital_intputs_60FD;
	::AWOpen:tyParamOutDriver.siModOfOpt_6060 AT %QB."AutoWidth".Modes_of_operation_6060;
	::AWOpen:tyParamOutDriver.diTargetPos_607A AT %QD."AutoWidth".Target_position_607A;
	::AWOpen:tyParamOutDriver.udiMoveSpd_6081 AT %QD."AutoWidth".Profile_velocity_6081;
	::AWOpen:tyParamOutDriver.siHmMethod_6098 AT %QB."AutoWidth".Homing_method_6098;
	::AWOpen:tyParamOutDriver.diJogVel_60FF AT %QD."AutoWidth".Target_velocity_60FF;
	::LifterBtm:tyParamInDriver.uiErrCode_603F AT %IW."Lifter".Error_code_603F;
	::LifterBtm:tyParamInDriver.siModOfOptDisp_6061 AT %IB."Lifter".Modes_of_operation_display_6061;
	::LifterBtm:tyParamInDriver.diActualPos_6064 AT %ID."Lifter".Position_actual_value_6064;
	::LifterBtm:tyParamInDriver.udiDigitalInputs_60FD AT %ID."Lifter".Digital_intputs_60FD;
	::LifterBtm:tyParamOutDriver.siModOfOpt_6060 AT %QB."Lifter".Modes_of_operation_6060;
	::LifterBtm:tyParamOutDriver.diTargetPos_607A AT %QD."Lifter".Target_position_607A;
	::LifterBtm:tyParamOutDriver.udiMoveSpd_6081 AT %QD."Lifter".Profile_velocity_6081;
	::LifterBtm:tyParamOutDriver.siHmMethod_6098 AT %QB."Lifter".Homing_method_6098;
	::LifterBtm:tyParamOutDriver.diJogVel_60FF AT %QD."Lifter".Target_velocity_60FF;
	::MagAWOpen1:tyParamInDriver.uiErrCode_603F AT %IW."Mag1_AutoWidth".Error_code_603F;
	::MagAWOpen1:tyParamInDriver.siModOfOptDisp_6061 AT %IB."Mag1_AutoWidth".Modes_of_operation_display_6061;
	::MagAWOpen1:tyParamInDriver.diActualPos_6064 AT %ID."Mag1_AutoWidth".Position_actual_value_6064;
	::MagAWOpen1:tyParamInDriver.udiDigitalInputs_60FD AT %ID."Mag1_AutoWidth".Digital_intputs_60FD;
	::MagAWOpen1:tyParamOutDriver.siModOfOpt_6060 AT %QB."Mag1_AutoWidth".Modes_of_operation_6060;
	::MagAWOpen1:tyParamOutDriver.diTargetPos_607A AT %QD."Mag1_AutoWidth".Target_position_607A;
	::MagAWOpen1:tyParamOutDriver.udiMoveSpd_6081 AT %QD."Mag1_AutoWidth".Profile_velocity_6081;
	::MagAWOpen1:tyParamOutDriver.siHmMethod_6098 AT %QB."Mag1_AutoWidth".Homing_method_6098;
	::MagAWOpen1:tyParamOutDriver.diJogVel_60FF AT %QD."Mag1_AutoWidth".Target_velocity_60FF;
	::MagAWOpen2:tyParamInDriver.uiErrCode_603F AT %IW."Mag2_AutoWidth".Error_code_603F;
	::MagAWOpen2:tyParamInDriver.siModOfOptDisp_6061 AT %IB."Mag2_AutoWidth".Modes_of_operation_display_6061;
	::MagAWOpen2:tyParamInDriver.diActualPos_6064 AT %ID."Mag2_AutoWidth".Position_actual_value_6064;
	::MagAWOpen2:tyParamInDriver.udiDigitalInputs_60FD AT %ID."Mag2_AutoWidth".Digital_intputs_60FD;
	::MagAWOpen2:tyParamOutDriver.siModOfOpt_6060 AT %QB."Mag2_AutoWidth".Modes_of_operation_6060;
	::MagAWOpen2:tyParamOutDriver.diTargetPos_607A AT %QD."Mag2_AutoWidth".Target_position_607A;
	::MagAWOpen2:tyParamOutDriver.udiMoveSpd_6081 AT %QD."Mag2_AutoWidth".Profile_velocity_6081;
	::MagAWOpen2:tyParamOutDriver.siHmMethod_6098 AT %QB."Mag2_AutoWidth".Homing_method_6098;
	::MagAWOpen2:tyParamOutDriver.diJogVel_60FF AT %QD."Mag2_AutoWidth".Target_velocity_60FF;
	::MagAWOpen3:tyParamInDriver.uiErrCode_603F AT %IW."Mag3_AutoWidth".Error_code_603F;
	::MagAWOpen3:tyParamInDriver.siModOfOptDisp_6061 AT %IB."Mag3_AutoWidth".Modes_of_operation_display_6061;
	::MagAWOpen3:tyParamInDriver.diActualPos_6064 AT %ID."Mag3_AutoWidth".Position_actual_value_6064;
	::MagAWOpen3:tyParamInDriver.udiDigitalInputs_60FD AT %ID."Mag3_AutoWidth".Digital_intputs_60FD;
	::MagAWOpen3:tyParamOutDriver.siModOfOpt_6060 AT %QB."Mag3_AutoWidth".Modes_of_operation_6060;
	::MagAWOpen3:tyParamOutDriver.diTargetPos_607A AT %QD."Mag3_AutoWidth".Target_position_607A;
	::MagAWOpen3:tyParamOutDriver.udiMoveSpd_6081 AT %QD."Mag3_AutoWidth".Profile_velocity_6081;
	::MagAWOpen3:tyParamOutDriver.siHmMethod_6098 AT %QB."Mag3_AutoWidth".Homing_method_6098;
	::MagAWOpen3:tyParamOutDriver.diJogVel_60FF AT %QD."Mag3_AutoWidth".Target_velocity_60FF;
	::AWPushOrPu:tyParamOutDriver.siModOfOpt_6060 AT %QB."AutoWidthPusher".Modes_of_operation_6060;
	::AWPushOrPu:tyParamOutDriver.diTargetPos_607A AT %QD."AutoWidthPusher".Target_position_607A;
	::AWPushOrPu:tyParamOutDriver.udiMoveSpd_6081 AT %QD."AutoWidthPusher".Profile_velocity_6081;
	::AWPushOrPu:tyParamOutDriver.siHmMethod_6098 AT %QB."AutoWidthPusher".Homing_method_6098;
	::AWPushOrPu:tyParamOutDriver.diJogVel_60FF AT %QD."AutoWidthPusher".Target_velocity_60FF;
	::AWPushOrPu:tyParamInDriver.uiErrCode_603F AT %IW."AutoWidthPusher".Error_code_603F;
	::AWPushOrPu:tyParamInDriver.siModOfOptDisp_6061 AT %IB."AutoWidthPusher".Modes_of_operation_display_6061;
	::AWPushOrPu:tyParamInDriver.diActualPos_6064 AT %ID."AutoWidthPusher".Position_actual_value_6064;
	::AWPushOrPu:tyParamInDriver.udiDigitalInputs_60FD AT %ID."AutoWidthPusher".Digital_intputs_60FD;
	::Trav:bModuleOK AT %IX."Traverser".ModuleOk;
	::Trav:tyParamInDriver.uiErrCode_603F AT %IW."Traverser".Error_code_603F;
	::Trav:tyParamInDriver.uiStatword_6041 AT %IW."Traverser".Statusword_6041;
	::Trav:tyParamInDriver.siModOfOptDisp_6061 AT %IB."Traverser".Modes_of_operation_display_6061;
	::Trav:tyParamInDriver.diActualPos_6064 AT %ID."Traverser".Position_actual_value_6064;
	::Trav:tyParamInDriver.udiDigitalInputs_60FD AT %ID."Traverser".Digital_intputs_60FD;
	::Trav:tyParamOutDriver.uiCtrlword_6040 AT %QW."Traverser".Controlword_6040;
	::Trav:tyParamOutDriver.siModOfOpt_6060 AT %QB."Traverser".Modes_of_operation_6060;
	::Trav:tyParamOutDriver.diTargetPos_607A AT %QD."Traverser".Target_position_607A;
	::Trav:tyParamOutDriver.udiMoveSpd_6081 AT %QD."Traverser".Profile_velocity_6081;
	::Trav:tyParamOutDriver.siHmMethod_6098 AT %QB."Traverser".Homing_method_6098;
	::Trav:tyParamOutDriver.diJogVel_60FF AT %QD."Traverser".Target_velocity_60FF;
	::PullerPush:bModuleOK AT %IX."PullerPusher".ModuleOk;
	::PullerPush:tyParamInDriver.uiErrCode_603F AT %IW."PullerPusher".ErrorCode_603F;
	::PullerPush:tyParamInDriver.uiStatword_6041 AT %IW."PullerPusher".Statusword_6041;
	::PullerPush:tyParamInDriver.siModOfOptDisp_6061 AT %IB."PullerPusher".ModesOfOperationDisplay_6061;
	::PullerPush:tyParamInDriver.udiDigitalInputs_60FD AT %ID."PullerPusher".DigitalInputs_60FD;
	::PullerPush:tyParamOutDriver.uiCtrlword_6040 AT %QW."PullerPusher".Controlword_6040;
	::PullerPush:tyParamOutDriver.siModOfOpt_6060 AT %QB."PullerPusher".ModesOfOperation_6060;
	::PullerPush:tyParamInDriver.diActualPos_6064 AT %ID."PullerPusher".PositionActualValue_6064;
	::PullerPush:tyParamOutDriver.diTargetPos_607A AT %QD."PullerPusher".TargetPosition_607A;
	::PullerPush:tyParamOutDriver.udiMoveSpd_6081 AT %QD."PullerPusher".ProfileVelocity_6081;
	::PullerPush:tyParamOutDriver.siHmMethod_6098 AT %QB."PullerPusher".HomingMethod_6098;
	::PullerPush:tyParamOutDriver.diJogVel_60FF AT %QD."PullerPusher".TargetVelocity_60FF;
	::Trav:tyParamInDriver.uiErrCode_603F AT %IW."Traverser".ErrorCode_603F;
	::Trav:tyParamOutDriver.siModOfOpt_6060 AT %QB."Traverser".ModesOfOperation_6060;
	::Trav:tyParamOutDriver.diTargetPos_607A AT %QD."Traverser".TargetPosition_607A;
	::Trav:tyParamOutDriver.udiMoveSpd_6081 AT %QD."Traverser".ProfileVelocity_6081;
	::Trav:tyParamOutDriver.siHmMethod_6098 AT %QB."Traverser".HomingMethod_6098;
	::Trav:tyParamOutDriver.diJogVel_60FF AT %QD."Traverser".TargetVelocity_60FF;
	::Trav:tyParamInDriver.siModOfOptDisp_6061 AT %IB."Traverser".ModesOfOperationDisplay_6061;
	::Trav:tyParamInDriver.diActualPos_6064 AT %ID."Traverser".PositionActualValue_6064;
	::Trav:tyParamInDriver.udiDigitalInputs_60FD AT %ID."Traverser".DigitalInputs_60FD;
	::AWOpen:bModuleOK AT %IX."AutoWidth_1".ModuleOk;
	::AWOpen:tyParamInDriver.uiErrCode_603F AT %IW."AutoWidth_1".Error_code_603F;
	::AWOpen:tyParamInDriver.uiStatword_6041 AT %IW."AutoWidth_1".Statusword_6041;
	::AWOpen:tyParamInDriver.siModOfOptDisp_6061 AT %IB."AutoWidth_1".Modes_of_operation_display_6061;
	::AWOpen:tyParamInDriver.diActualPos_6064 AT %ID."AutoWidth_1".Position_actual_value_6064;
	::AWOpen:tyParamInDriver.udiDigitalInputs_60FD AT %ID."AutoWidth_1".Digital_intputs_60FD;
	::AWOpen:tyParamOutDriver.uiCtrlword_6040 AT %QW."AutoWidth_1".Controlword_6040;
	::AWOpen:tyParamOutDriver.siModOfOpt_6060 AT %QB."AutoWidth_1".Modes_of_operation_6060;
	::AWOpen:tyParamOutDriver.diTargetPos_607A AT %QD."AutoWidth_1".Target_position_607A;
	::AWOpen:tyParamOutDriver.udiMoveSpd_6081 AT %QD."AutoWidth_1".Profile_velocity_6081;
	::AWOpen:tyParamOutDriver.siHmMethod_6098 AT %QB."AutoWidth_1".Homing_method_6098;
	::AWOpen:tyParamOutDriver.diJogVel_60FF AT %QD."AutoWidth_1".Target_velocity_60FF;
	::LifterBtm:bModuleOK AT %IX."Lifter_2".ModuleOk;
	::LifterBtm:tyParamInDriver.uiErrCode_603F AT %IW."Lifter_2".Error_code_603F;
	::LifterBtm:tyParamInDriver.uiStatword_6041 AT %IW."Lifter_2".Statusword_6041;
	::LifterBtm:tyParamInDriver.siModOfOptDisp_6061 AT %IB."Lifter_2".Modes_of_operation_display_6061;
	::LifterBtm:tyParamInDriver.diActualPos_6064 AT %ID."Lifter_2".Position_actual_value_6064;
	::LifterBtm:tyParamInDriver.udiDigitalInputs_60FD AT %ID."Lifter_2".Digital_intputs_60FD;
	::LifterBtm:tyParamOutDriver.uiCtrlword_6040 AT %QW."Lifter_2".Controlword_6040;
	::LifterBtm:tyParamOutDriver.siModOfOpt_6060 AT %QB."Lifter_2".Modes_of_operation_6060;
	::LifterBtm:tyParamOutDriver.diTargetPos_607A AT %QD."Lifter_2".Target_position_607A;
	::LifterBtm:tyParamOutDriver.udiMoveSpd_6081 AT %QD."Lifter_2".Profile_velocity_6081;
	::LifterBtm:tyParamOutDriver.siHmMethod_6098 AT %QB."Lifter_2".Homing_method_6098;
	::LifterBtm:tyParamOutDriver.diJogVel_60FF AT %QD."Lifter_2".Target_velocity_60FF;
	::Trav:bModuleOK AT %IX."Traverser_1".ModuleOk;
	::Trav:tyParamInDriver.uiErrCode_603F AT %IW."Traverser_1".Error_code_603F;
	::Trav:tyParamInDriver.uiStatword_6041 AT %IW."Traverser_1".Statusword_6041;
	::Trav:tyParamInDriver.siModOfOptDisp_6061 AT %IB."Traverser_1".Modes_of_operation_display_6061;
	::Trav:tyParamInDriver.diActualPos_6064 AT %ID."Traverser_1".Position_actual_value_6064;
	::Trav:tyParamInDriver.udiDigitalInputs_60FD AT %ID."Traverser_1".Digital_intputs_60FD;
	::Trav:tyParamOutDriver.uiCtrlword_6040 AT %QW."Traverser_1".Controlword_6040;
	::Trav:tyParamOutDriver.siModOfOpt_6060 AT %QB."Traverser_1".Modes_of_operation_6060;
	::Trav:tyParamOutDriver.diTargetPos_607A AT %QD."Traverser_1".Target_position_607A;
	::Trav:tyParamOutDriver.udiMoveSpd_6081 AT %QD."Traverser_1".Profile_velocity_6081;
	::Trav:tyParamOutDriver.siSchHmMethod_6098 AT %QB."Traverser_1".Homing_method_6098;
	::Trav:tyParamOutDriver.diJogVel_60FF AT %QD."Traverser_1".Target_velocity_60FF;
END_VAR
```

## Configuration 3Mag_UL_SOT_Estun_MPuller

CPU X20CP0483, AutomationRuntime B4.82, Build 4.1.2, Safety 0.0, Vc V4.72.1

### Task classes (Cpu.sw)
```
Cyclic#1 (cycle 10000 us, tolerance 10000 us):
  DInput <- DInput.DInput.prg
  DOutput <- DOutput.DOutput.prg
Cyclic#2 (cycle 20000 us, tolerance 20000 us):
  PshrConv <- Conv.PshrConv.prg
  MagConv2Cl <- MagConv_LiftnTrav.MagConv2Clp1.prg
  MagConv2C1 <- MagConv_LiftnTrav.MagConv2Clp2.prg
  MagConv2C2 <- MagConv_LiftnTrav.MagConv2Clp3.prg
Cyclic#3 (cycle 50000 us, tolerance 50000 us):
  UI <- UI.UI.prg
  Startup <- Startup.Startup.prg
  General <- General.General.prg
  UsrFolder <- UsrFolder.UsrFolder.prg
  LibVer <- LibVer.LibVer.prg
  HWInfo <- HWInfo.HWInfo.prg
  TLBuz <- TLBuz.TLBuz.prg
  Alarm <- Alarm.Alarm.prg
  ProdRcp <- ProdRcp.ProdRcp.prg
  MpProdRcp <- MpProdRcp.MpProdRcp.prg
  MagRcp <- MagRcp.MagRcp.prg
  McParam <- McParam.McParam.prg
  NtParam <- NtParam.NtParam.prg
  UsrMgmt <- UsrMgmt.UsrMgmt.prg
  OvenInfoA <- OvenInfo.OvenInfoA.prg
  OvenInfoB <- OvenInfo.OvenInfoB.prg
  Buffer1 <- Buffer.Buffer1.prg
  Buffer2 <- Buffer.Buffer2.prg
  Buffer3 <- Buffer.Buffer3.prg
  BufferMagA <- Buffer.BufferMagA.prg
  BufferMagB <- Buffer.BufferMagB.prg
  USSMEMAA <- SMEMA.USSMEMAA.prg
  USSMEMAB <- SMEMA.USSMEMAB.prg
  USSMEMA1 <- SMEMA.USSMEMA1.prg
  USSMEMA2 <- SMEMA.USSMEMA2.prg
  USSMEMA3 <- SMEMA.USSMEMA3.prg
  DSSMEMA1 <- SMEMA.DSSMEMA1.prg
  DSSMEMA2 <- SMEMA.DSSMEMA2.prg
  DSSMEMA3 <- SMEMA.DSSMEMA3.prg
  Pneu2SenIn <- Pneu.PneuInShutter.prg
  Pneu2SenOu <- Pneu.PneuOutShutter.prg
  PneuNoSenS <- Pneu.PneuStopperA.prg
  PneuNoSen1 <- Pneu.PneuStopperB.prg
  AWPushOrPu <- CANOpenServo.AW.AWPushOrPuller.prg
  AWOpen <- CANOpenServo.AW.AWOpen.prg
  Trav <- CANOpenServo.Trav.Trav.prg
  LifterBtm <- CANOpenServo.Lifter.LifterBtm.prg
  LFLeader <- LF.LFLeader.prg
  LFFollower <- LF.LFFollower.prg
  Follower1 <- LF.Follower1.prg
  Follower2 <- LF.Follower2.prg
  LCS <- LCS.LCS.prg
  LCSMngRcp <- LCS.LCSMngRcp.prg
  LCSLF <- LCS.LCSLF.prg
  Ops <- Operations.Ops.prg
  OpsTravLif <- Operations.OpsTravLifUL.prg
  OpsMagConv <- Operations.MagConv_StationaryPlat.OpsMagConvUL1.prg
  OpsMagCon1 <- Operations.MagConv_StationaryPlat.OpsMagConvUL2.prg
  OpsMagCon2 <- Operations.MagConv_StationaryPlat.OpsMagConvUL3.prg
  OpsLifMagU <- Operations.OpsLifMagUL.prg
  Pneu2SenSe <- Pneu.PneuSelClamp1.prg
  AGV <- AGVCom.AGV.prg
  AGV1 <- AGVCom.AGV1.prg
  AGV2 <- AGVCom.AGV2.prg
  AGV3 <- AGVCom.AGV3.prg
  Simu <- Simulation.Simu.prg
  Simu1 <- Simulation.Simu.prg
  Machine <- Machine.Machine.prg
  MagAWOpen1 <- CANOpenServo.MagAW.MagAWOpen1.prg
  MagAWOpen2 <- CANOpenServo.MagAW.MagAWOpen2.prg
  MagAWOpen3 <- CANOpenServo.MagAW.MagAWOpen3.prg
  Pneu2SenMa <- Pneu.PneuMag1SafetyBar.prg
  Pneu2SenM3 <- Pneu.PneuMag1AWEngage.prg
  USSOT1 <- SOT.USSOT1.prg
  DSSOT1 <- SOT.DSSOT1.prg
  MtrPshr <- MtrPshr.MtrPshr.prg
Cyclic#4 (cycle 10000 us, tolerance 10000 us):
  PullerPush <- CANOpenServo.PullerPusher.PullerPusher.prg
  Hermes <- Hermes.Hermes.prg
  USHermesA <- Hermes.USHermesA.prg
  USHermesB <- Hermes.USHermesB.prg
  RmtHermes <- Hermes.RmtHermes.prg
  SvyHermes <- Hermes.SvyHermes.prg
  RstErr <- RstErr.RstErr.prg
DataObjects: Acp10sys
VcDataObjects: Visu <- UI.Visu.dob
Binaries: vcfntttf, arialbi, vccbmp, vcshared, vcpdvnc, vccshape, vcfile, vcgclass, arial, vcchspot, vcmgr, arialxsr, vccslider, vcdsint, vccbtn, vcdsloc, vccovl, vccpopup, vccline, vcctext, vcalarm, vcbclass, vccbar, visvc, udbdef, vcrt, vccnum, vccstr, Visu03, vccddbox, arialbd, vcpdsw, vcnet, TCData, Visu02, Visu01, vctcal, vccdt, arsvcreg, vcpfgen, acp10cfg, Acp10map, arconfig, asfw, iomap, Role, ashwd, ashwac, sysconf, User, Config, vcpfar00, OpcUaMap
Libraries: AsOpcUac, sys_lib, asstring, visapi, AsMem, astime, AsCANopen, AsIecCon, AsIODiag, FileIO, AsTCP, runtime, standard, brsystem, AsFltGen, dvframe, MpRecipe, MpBase, MpCom, NtBuffer, NtConv, NtFileIO, NtLogFile, NtMem, NtMessage, NtOvenInfo, NtPneu, NtRS232, NtSMEMA, NtTCP, NtTLBuz, NtVersion, NtSOT, vcresman, dataobj, asarcfg, powerlnk, NtGeneral, NtUI, NtHermes, NtOpConXML
```

### Hardware
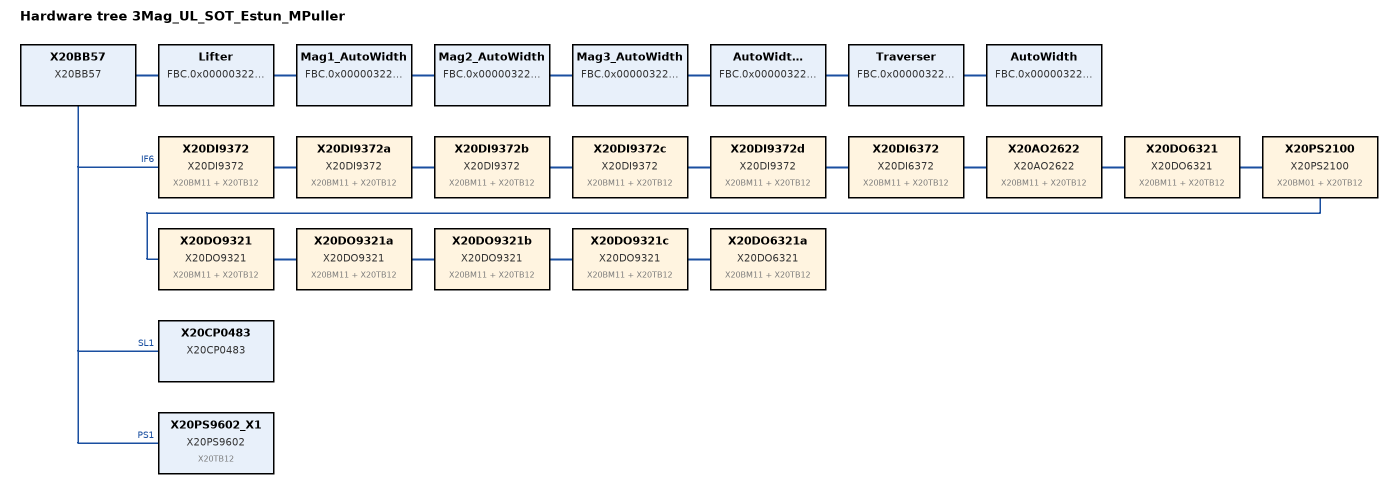
```
AutoWidth : FBC.0x00000322.0x00001000.NUTEK_ESTUN_PronetPlus_EDS_V106 v1.06.1 (OrderNumber=NUTEK_ESTUN_PronetPlus_V106)  [CAN1 -> Traverser.CAN2 (NodeNumber=16)]
AutoWidthPusher : FBC.0x00000322.0x00001000.NUTEK_ESTUN_PronetPlus_EDS_V106 v1.06.1 (OrderNumber=NUTEK_ESTUN_PronetPlus_V106)  [CAN1 -> Mag3_AutoWidth.CAN2]
Lifter : FBC.0x00000322.0x00001000.NUTEK_ESTUN_PronetPlus_EDS_V106 v1.06.1 (OrderNumber=NUTEK_ESTUN_PronetPlus_V106)  [CAN1 -> X20BB57.IF7 (NodeNumber=17)]
Mag1_AutoWidth : FBC.0x00000322.0x00001000.NUTEK_ESTUN_PronetPlus_EDS_V106 v1.06.1 (OrderNumber=NUTEK_ESTUN_PronetPlus_V106)  [CAN1 -> Lifter.CAN2 (NodeNumber=19)]
Mag2_AutoWidth : FBC.0x00000322.0x00001000.NUTEK_ESTUN_PronetPlus_EDS_V106 v1.06.1 (OrderNumber=NUTEK_ESTUN_PronetPlus_V106)  [CAN1 -> Mag1_AutoWidth.CAN2]
Mag3_AutoWidth : FBC.0x00000322.0x00001000.NUTEK_ESTUN_PronetPlus_EDS_V106 v1.06.1 (OrderNumber=NUTEK_ESTUN_PronetPlus_V106)  [CAN1 -> Mag2_AutoWidth.CAN2]
Traverser : FBC.0x00000322.0x00001000.NUTEK_ESTUN_PronetPlus_EDS_V106 v1.06.1 (OrderNumber=NUTEK_ESTUN_PronetPlus_V106)  [CAN1 -> AutoWidthPusher.CAN2 (NodeNumber=18)]
X20AO2622 : X20AO2622 v1.2.0.0  [SS1 -> X20TB12m.SS; SL -> X20BM11k.SL1]
  Supervision = off
X20BB57 : X20BB57 v1.1.1.0
  Connector IF1:
    Baudrate = 9600
    Parity = N
  Connector IF7:
    Baudrate = 1000000
    ActivateCanOpen = 1
    p100c_parametervalue = 1000
    p100d_parametervalue = 3
X20BM01 : X20BM01 v2.1.0.0  [X2X1 -> X20BM11e.X2X2]
X20BM11 : X20BM11 v1.0.0.1  [X2X1 -> X20BB57.IF6]
X20BM11a : X20BM11 v1.0.0.1  [X2X1 -> X20BM11.X2X2]
X20BM11b : X20BM11 v1.0.0.1  [X2X1 -> X20BM11a.X2X2]
X20BM11c : X20BM11 v1.0.0.1  [X2X1 -> X20BM11b.X2X2]
X20BM11d : X20BM11 v1.0.0.1  [X2X1 -> X20BM11c.X2X2]
X20BM11e : X20BM11 v1.0.0.1  [X2X1 -> X20BM11k.X2X2]
X20BM11f : X20BM11 v1.0.0.1  [X2X1 -> X20BM01.X2X2]
X20BM11g : X20BM11 v1.0.0.1  [X2X1 -> X20BM11f.X2X2]
X20BM11h : X20BM11 v1.0.0.1  [X2X1 -> X20BM11g.X2X2]
X20BM11i : X20BM11 v1.0.0.1  [X2X1 -> X20BM11d.X2X2]
X20BM11j : X20BM11 v1.0.0.1  [X2X1 -> X20BM11h.X2X2]
X20BM11k : X20BM11 v1.0.0.1  [X2X1 -> X20BM11i.X2X2]
X20BM11l : X20BM11 v1.0.0.1  [X2X1 -> X20BM11j.X2X2]
X20CP0483 : X20CP0483 v1.2.1.0  [SL -> X20BB57.SL1]
  Connector IF2:
    ActivateDevice = 1
    Mode = Manual
    InternetAddress = 192.168.0.24
    SubnetMask = 255.255.255.0
    InaNodeNumber = 24
    Vnc1
    VncVcObjectName1 = Visu
    VncKeyMappingFile1 = 
    VncMaxConnections1 = 3
    VncRefreshRate1 = 100
    ActivateSnmp = 2
  ConfigurationID = NAEUL004
  VolatileGlobalPvSize = 80000
  EnableUsbRemoteInstall = 1
  TimerDeviceType = SWIOTIMER
  Cyclic1Duration = 10000
  Cyclic1Tolerance = 10000
  Cyclic2Duration = 20000
  Cyclic2Tolerance = 20000
  Cyclic3Duration = 50000
  Cyclic3Tolerance = 50000
  Cyclic4Duration = 10000
  Cyclic4Tolerance = 10000
  Cyclic5Duration = 200000
  Cyclic5Tolerance = 200000
  Cyclic6Duration = 500000
  Cyclic6Tolerance = 500000
  Cyclic7Duration = 1000000
  Cyclic7Tolerance = 1000000
  Cyclic8Duration = 10000
  Cyclic8Tolerance = 10000
  FileDevice1
  FileDeviceName1 = C
  FileDevicePath1 = C:
  FileDevice2
  FileDeviceName2 = User
  FileDevicePath2 = C:\User
  FileDevice3
  FileDeviceName3 = Private
  FileDevicePath3 = C:\Private
  FileDevice4
  FileDeviceName4 = CustomerUser
  FileDevicePath4 = C:\User\UserMgmt
  FileDevice5
  FileDeviceName5 = ProdRcp
  FileDevicePath5 = C:\User\ProductRecipe
  FileDevice6
  FileDeviceName6 = MagRcp
  FileDevicePath6 = C:\User\MagazineRecipe
  FileDevice7
  FileDeviceName7 = Alarm
  FileDevicePath7 = C:\User\Alarm
  FileDevice8
  FileDeviceName8 = McParam
  FileDevicePath8 = C:\User\MachineParameter
  FileDevice9
  FileDeviceName9 = NtParam
  FileDevicePath9 = C:\Private\NutekParameter
  FileDevice10
  FileDeviceName10 = LibVer
  FileDevicePath10 = C:\User\LibrariesVersion
  FileDevice11
  FileDeviceName11 = Retain
  FileDevicePath11 = C:\User\Retain
  FileDevice12
  FileDeviceName12 = Log
  FileDevicePath12 = C:\User\Log
  FileDevice13
  FileDeviceName13 = LCS
  FileDevicePath13 = C:\User\LCS
  FileDevice14
  FileDeviceName14 = MpProdRcp
  FileDevicePath14 = C:\User\ProductRecipeXml
  FileDevice15
  FileDeviceName15 = MpNtParam
  FileDevicePath15 = C:\Private\NutekParameterXml
  FtpUser1
  FtpUsername1 = NTAFTP
  FtpUserPassword1 = +UZ5u8Axw7KkkY4oM/r7wOOfB5oWHxpSY6r3j++jJso=  // NTA4BH
  FtpUserSalt1 = c0Alfi1W
  FTPAccessRight1 = 0
  FTPdevice1 = ALL
  FtpUser2
  FtpUsername2 = admin
  FtpUserPassword2 = mW+qRsE1LOSFDAB60rBJwb9dZ7uQUIuoHZp04C+x5XU=  // admin
  FtpUserSalt2 = Nr9+IHjr
  FTPAccessRight2 = 0
  FTPMSPartition2 = SYSTEM
  FTPMSpath2 = User
  FtpUser3
  FtpUsername3 = LCS
  FtpUserPassword3 = W4lkF6NjcyaB1sRdLwIoSAlqHoAE4GimWQdq7pKTzbA=  // LCS
  FtpUserSalt3 = f3H7b7h0
  FTPMSPartition3 = SYSTEM
  FTPMSpath3 = User\LCS
  ActivateOpcUa = 1
  OpcUa_ConversationSecurityPolicy_EnableBasic256Rsa256 = 0
  OpcUaInformationModels_PV_Version = 1
X20DI6372 : X20DI6372 v1.1.0.0  [SS1 -> X20TB12k.SS; SL -> X20BM11i.SL1]
  Supervision = off
X20DI9372 : X20DI9372 v1.1.0.0  [SS1 -> X20TB12a.SS; SL -> X20BM11.SL1]
  Supervision = off
X20DI9372a : X20DI9372 v1.1.0.0  [SS1 -> X20TB12b.SS; SL -> X20BM11a.SL1]
  Supervision = off
X20DI9372b : X20DI9372 v1.1.0.0  [SS1 -> X20TB12c.SS; SL -> X20BM11b.SL1]
  Supervision = off
X20DI9372c : X20DI9372 v1.1.0.0  [SS1 -> X20TB12d.SS; SL -> X20BM11c.SL1]
  Supervision = off
X20DI9372d : X20DI9372 v1.1.0.0  [SS1 -> X20TB12e.SS; SL -> X20BM11d.SL1]
  Supervision = off
X20DO6321 : X20DO6321 v1.1.0.0  [SS1 -> X20TB12f.SS; SL -> X20BM11e.SL1]
  Supervision = off
X20DO6321a : X20DO6321 v1.1.0.0  [SS1 -> X20TB12n.SS; SL -> X20BM11l.SL1]
  Supervision = off
X20DO9321 : X20DO9321 v1.1.0.0  [SS1 -> X20TB12h.SS; SL -> X20BM11f.SL1]
  Supervision = off
X20DO9321a : X20DO9321 v1.1.0.0  [SS1 -> X20TB12i.SS; SL -> X20BM11g.SL1]
  Supervision = off
X20DO9321b : X20DO9321 v1.1.0.0  [SS1 -> X20TB12j.SS; SL -> X20BM11h.SL1]
  Supervision = off
X20DO9321c : X20DO9321 v1.1.0.0  [SS1 -> X20TB12l.SS; SL -> X20BM11j.SL1]
  Supervision = off
X20PS2100 : X20PS2100 v1.2.0.0  [SS1 -> X20TB12g.SS; SL -> X20BM01.SL1]
  Supervision = off
X20PS9602_X1 : X20PS9602 v1.0.2.0  [PS -> X20BB57.PS1; SS1 -> X20TB12.SS]
X20TB12 : X20TB12 v1.0.0.0
X20TB12a : X20TB12 v1.0.0.0
X20TB12b : X20TB12 v1.0.0.0
X20TB12c : X20TB12 v1.0.0.0
X20TB12d : X20TB12 v1.0.0.0
X20TB12e : X20TB12 v1.0.0.0
X20TB12f : X20TB12 v1.0.0.0
X20TB12g : X20TB12 v1.0.0.0
X20TB12h : X20TB12 v1.0.0.0
X20TB12i : X20TB12 v1.0.0.0
X20TB12j : X20TB12 v1.0.0.0
X20TB12k : X20TB12 v1.0.0.0
X20TB12l : X20TB12 v1.0.0.0
X20TB12m : X20TB12 v1.0.0.0
X20TB12n : X20TB12 v1.0.0.0
```
